(******ErrorStatus******)
IF axisdata[4].Axis_Error OR axisdata[5].Axis_Error THEN
	FeedIndexer.ErrorStatus.errErrorActive:=1;
ELSE
	FeedIndexer.ErrorStatus.errErrorActive:=0;
END_IF
FeedIndexer.ErrorStatus.errFieldBus:=0;
FeedIndexer.ErrorStatus.errLim2CCW:=b_limit_final_ccw_FI;
FeedIndexer.ErrorStatus.errLim2CW:=b_limit_final_cw_FI;
IF status_code4 = 'E2059' OR status_code5 = 'E2059' THEN
	FeedIndexer.ErrorStatus.errLimV_Err:=1;
ELSE
	FeedIndexer.ErrorStatus.errLimV_Err:=0;
END_IF
FeedIndexer.ErrorStatus.errMotComm:=(NOT(axisdata[4].Axis_NRT) OR NOT(axisdata[5].Axis_NRT));
IF status_code4 = 'F2031' OR status_code5 = 'F2031' THEN
	FeedIndexer.ErrorStatus.errMotEnc:=1;
ELSE
	FeedIndexer.ErrorStatus.errMotEnc:=0;
END_IF
IF status_code4 = 'F2021' OR status_code5 = 'F2021' OR FeedIndexer.ErrorStatus.errMotEnc THEN
	FeedIndexer.ErrorStatus.errMotor:=1;
ELSE
	FeedIndexer.ErrorStatus.errMotor:=0;
END_IF
IF FeedIndexer.ErrorStatus.errMotor OR FeedIndexer.ErrorStatus.errMotEnc THEN
	FeedIndexer.ErrorStatus.errMotReady:=1;
ELSE
	FeedIndexer.ErrorStatus.errMotReady:=0;
END_IF
FeedIndexer.ErrorStatus.errOverride:=0;
FeedIndexer.ErrorStatus.errV_DevExceed:=FeedIndexer.ErrorStatus.errLimV_Err;
IF status_code4 = 'F2075' THEN
	FeedIndexer.ErrorStatus.errP_RangeExceed:=1;
ELSE
	FeedIndexer.ErrorStatus.errP_RangeExceed:=0;
END_IF
IF status_code4 = 'F2037' OR status_code5 = 'F2037' THEN
	FeedIndexer.ErrorStatus.errP_DevExceed:=1;
ELSE
	FeedIndexer.ErrorStatus.errP_DevExceed:=0;
END_IF
FeedIndexer.ErrorStatus.errPosEnc:=FeedIndexer.Status.encBoxOp;
FeedIndexer.ErrorStatus.errPosEnc_Fo:=FeedIndexer.Status.encBoxOp;
IF status_code4 = 'F2026' OR status_code5 = 'F2026' THEN
	FeedIndexer.ErrorStatus.errPower:=1;
ELSE
	FeedIndexer.ErrorStatus.errPower:=0;
END_IF
(***** Error status end*****)


(*******Warning state********)
FeedIndexer.WarningStatus.waLim1CW:=b_limit_cw_FI;
FeedIndexer.WarningStatus.waLim1CCW:=b_limit_ccw_FI;
IF status_code4 = 'E8029' OR status_code5 = 'E8029' THEN
	FeedIndexer.WarningStatus.waLimSoftCW:=1;
ELSE
	FeedIndexer.WarningStatus.waLimSoftCW:=0;
END_IF
IF status_code4 = 'E8030' OR status_code5 = 'E8030' THEN
	FeedIndexer.WarningStatus.waLimSoftCCW:=1;
ELSE
	FeedIndexer.WarningStatus.waLimSoftCCW:=0;
END_IF
IF status_code4 = 'E8260' OR status_code5 = 'E8260' THEN
	FeedIndexer.WarningStatus.waMmaxExceeded:=1;
ELSE
	FeedIndexer.WarningStatus.waMmaxExceeded:=0;
END_IF
FeedIndexer.WarningStatus.waMotReady:=FeedIndexer.ErrorStatus.errMotReady;
FeedIndexer.WarningStatus.waMotWarn:=(axisdata[4].Axis_Warning OR axisdata[4].Axis_Warning);
FeedIndexer.WarningStatus.waOverride:=0;
FeedIndexer.WarningStatus.waParamFault:=(FeedIndexer.WarningStatus.waMotReady OR FeedIndexer.ErrorStatus.errMotReady);
IF status_code4 = 'E2031' OR status_code5 = 'E2031' THEN
	FeedIndexer.WarningStatus.waPosEncWarn:=1;
ELSE
	FeedIndexer.WarningStatus.waPosEncWarn:=0;
END_IF
FeedIndexer.WarningStatus.waStowPinsDep:=FALSE;
FeedIndexer.WarningStatus.waVelLimit:=FeedIndexer.ErrorStatus.errV_DevExceed;
(*********Warning status end***********)
(*****motor1****)
FeedIndexer.MotorOne.ErrorCode:= STRING_TO_UINT(status_code4);
FeedIndexer.MotorOne.mActTorq:=r_torque_4*7.1;
FeedIndexer.MotorOne.mActVelocity:=i_speed_4;
FeedIndexer.MotorOne.MotorTemp:=r_temp_motor4;
FeedIndexer.MotorOne.RateOfUtil:=r_torque_4;
FeedIndexer.MotorOne.MotorOverload:=r_torque_4;
(*****motor2****)
FeedIndexer.MotorTwo.ErrorCode:= STRING_TO_UINT(status_code5);
FeedIndexer.MotorTwo.mActTorq:=r_torque_5*7.1;
FeedIndexer.MotorTwo.mActVelocity:=i_speed_5;
FeedIndexer.MotorTwo.MotorTemp:=r_temp_motor5;
FeedIndexer.MotorTwo.RateOfUtil:=r_torque_5;
FeedIndexer.MotorTwo.MotorOverload:=r_torque_5;

END_PROGRAM

// IndraMotionMlc1/Application/POUs/OPCUA/OPCUA_Node/P_Opcua_Safety
PROGRAM P_Opcua_Safety
VAR
	b_final_limit_active:BOOL;
	fb_move_stow_Az: MC_MoveAbsolute;
	fb_move_stow_El: MC_MoveAbsolute;
	fb_ton_stow: TON;
	fb_self_reset_stow: R_Trig;
	fb_ton_self_reset_stow: TON;
	fb_rtrig_off_stow:R_Trig;
	fb_rtrig_lock_stow: R_Trig;
	fb_rtrig_reset_deploy: R_Trig;
	fb_rtrig_reset_retract: R_Trig;
	fb_rtrig_estop: R_TRIG;
	fb_rtrig_interlock_Az: R_TRIG;
	fb_rtrig_interlock_El: R_TRIG;
	fb_rtrig_interlock_Fi: R_TRIG;
	
	fb_ton_sim_stow: TON;
	_retract: TON;
	fb_ton_sim_retract: TON;
	fb_ton_sim_deploy: TON;
	fb_rtrig_sim_retract: R_TRIG;
	fb_rtrig_sim_deploy: R_TRIG;
	fb_rtrig_stow_deactivate: R_TRIG;
	fb_rtrig_stow_pulse: R_TRIG;
	_test: BOOL;
	b_stow_SIP: BOOL;
	rtrig_Estop_Az: R_TRIG;
	fb_Estop_Az: MC_Stop;
	rtrig_Estop_El: R_TRIG;
	fb_Estop_El: MC_Stop;
	rtrig_Estop_Fi: R_TRIG;
	fb_Estop_Fi: MC_Stop;
	MC_MoveRelative_0: MC_MoveRelative;
	MC_MoveRelative_1: MC_MoveRelative;
	R_TRIG_0: R_TRIG;
	TON_0: TON;
	b_stow_wait: BOOL;
	TON_1: TON;
	b_stow_run: BOOL;
	R_TRIG_1: R_TRIG;
	F_TRIG_0: F_TRIG;
	F_TRIG_1: F_TRIG;
	F_TRIG_2: F_TRIG;
	F_TRIG_3: F_TRIG;
	F_TRIG_4: F_TRIG;
	fb_rtrig_deactivate_El: R_TRIG;
	fb_rtrig_clear_stow: R_TRIG;
	F_TRIG_5: F_trig;
END_VAR
VAR // added by the converter: edge detectors and wires of the graphical bodies
    _w1, _w2, _w3, _w4, _w5, _w6 : BOOL;
END_VAR

safety();
(*IF b_HHP_Estop OR b_Turnhead_Estop OR b_DS_Estop OR b_FI_Estop OR b_Turnhead_Hatch OR b_AZ_Hatch OR (NOT(b_stow_pin_limit_unlock)) THEN
	b_in_interlock:=1;
ELSE
	b_in_interlock:=0;
END_IF*)

(*IF b_in_interlock OR b_DSDoor_Estop OR b_PSCDoor_Estop OR b_DriveCabinetDoor_Estop OR b_EMISCDoor_Estop THEN // b_in_interlock true will cause an EStop. Whereas it should only cause an interlock. 
	b_in_Estop:=1;
ELSE
	b_in_Estop:=0;
END_IF*)
safety.Status.AutoStowActive:=0;
safety.Status.Axes_InitFault:=NOT(Azimuth.Status.InitOk AND Elevation.Status.InitOk AND FeedIndexer.Status.InitOk);
safety.Status.EStopFi:=b_FI_Estop;
safety.Status.EStopHHP:=b_HHP_Estop;
safety.Status.EStopPED:=b_DS_Estop;
safety.Status.EStopTurnhead:=b_Turnhead_Estop;
safety.Status.HatchTurnheadRoof:=b_Turnhead_Hatch;
safety.Status.HatchAzBearing:=b_AZ_Hatch;
//safety.InterlockAck
safety.Status.Lim2_CCW_Az:=b_limit_final_ccw_az;
safety.Status.Lim2_CCW_Fi:=b_limit_final_ccw_Fi;
safety.Status.Lim2_CW_Az:=b_limit_final_cw_az;
safety.Status.Lim2_CW_Fi:=b_limit_final_cw_Fi;
safety.Status.Lim2_Dn_El:=b_limit_final_ccw_el;
safety.Status.Lim2_Up_El:=b_limit_final_cw_el;
b_final_limit_active:=(safety.Status.Lim2_CCW_Az OR safety.Status.Lim2_CW_Az OR safety.Status.Lim2_Dn_El OR safety.Status.Lim2_Up_El OR safety.Status.Lim2_CCW_Fi OR safety.Status.Lim2_CW_Fi); 

(* Still to be wired in *)
safety.Status.SafetyLockout_Az:=NOT(b_Lock_Out_Az);
safety.Status.SafetyLockout_El:=NOT(b_Lock_Out_El);
safety.Status.SafetyLockout_Fi:=NOT(b_Lock_Out_Fi);

IF safety.Status.Axes_InitFault THEN
	safety.Status.SafetyState:=SafetyStatetype.Stopped;
ELSIF b_in_interlock OR b_in_Estop OR b_final_limit_active THEN
	safety.Status.SafetyState:=SafetyStatetype.Error;
ELSE
	safety.Status.SafetyState:=SafetyStatetype.Running;	
END_IF
safety.Status.STO_Az:=b_in_interlock;
safety.Status.STO_El:=b_in_interlock;
safety.Status.STO_Fi:=b_in_interlock;

IF b_stow_pin_deploy AND NOT(b_stow_pin_limit_lock) THEN
	safety.Status.StowPinStatus:=StowPinStatustype.Deploying;
ELSIF b_stow_pin_limit_lock THEN
	safety.Status.StowPinStatus:=StowPinStatustype.Deployed;
ELSIF b_stow_pin_retract AND NOT(b_stow_pin_limit_unlock) THEN
	safety.Status.StowPinStatus:=StowPinStatustype.Retracting;
ELSIF NOT(b_stow_pin_limit_unlock) THEN
	safety.Status.StowPinStatus:=StowPinStatustype.Retracted;
END_IF

IF (Azimuth.Status.p_Enc >= Azimuth.Status.StowPos_Minus AND Azimuth.Status.p_Enc <= Azimuth.Status.StowPos_Plus) THEN
	b_stow_lock_allow:=1;
ELSE 
	b_stow_lock_allow:=0;
END_IF

(*
IF b_in_interlock AND b_in_Estop THEN 
	Safety.Status.InterlockClearable:=0;
ELSE
	Safety.Status.InterlockClearable:=1;	
END_IF *)

// Run Ladder Logic
P_Opcua_Safety.A_STOW();
P_Opcua_Safety.A_Interlock_Estop();

ACTION A_STOW:
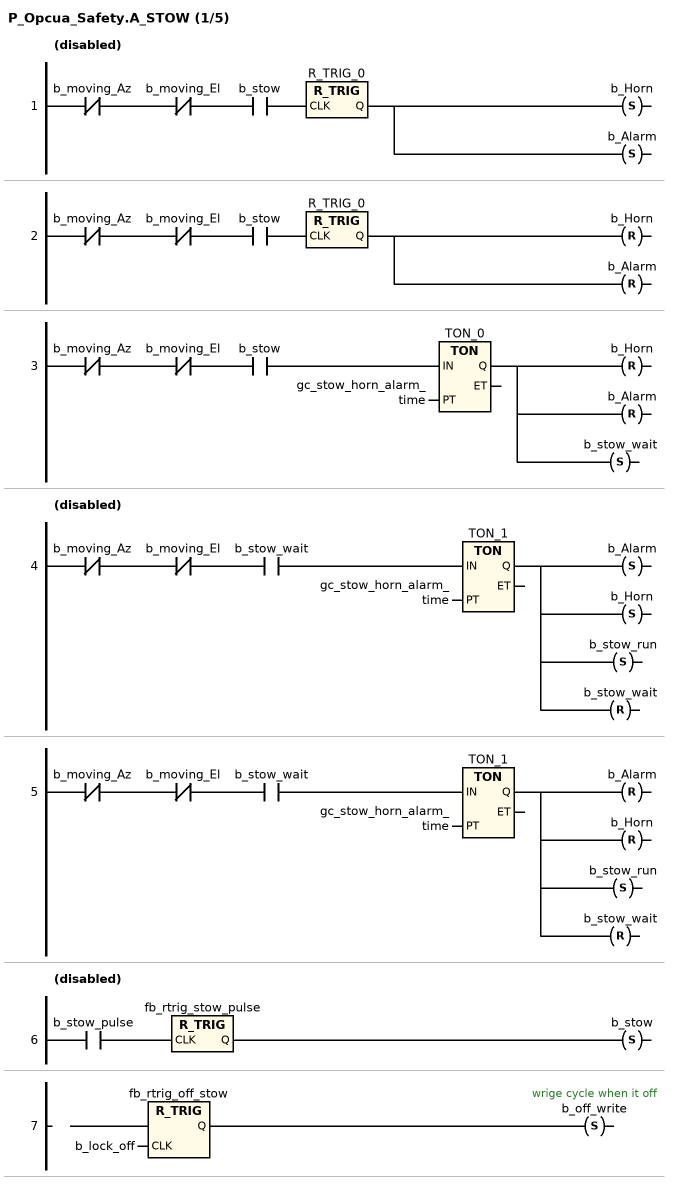
// NETWORK 1 (disabled)
// R_TRIG_0(CLK := NOT b_moving_Az AND NOT b_moving_El AND b_stow); // R_TRIG
// b_Horn S= R_TRIG_0.Q;
// b_Alarm S= R_TRIG_0.Q;

// NETWORK 2
R_TRIG_0(CLK := NOT b_moving_Az AND NOT b_moving_El AND b_stow); // R_TRIG
b_Horn R= R_TRIG_0.Q;
b_Alarm R= R_TRIG_0.Q;

// NETWORK 3
TON_0(IN := NOT b_moving_Az AND NOT b_moving_El AND b_stow, PT := gc_stow_horn_alarm_time); // TON
b_Horn R= TON_0.Q;
b_Alarm R= TON_0.Q;
b_stow_wait S= TON_0.Q;

// NETWORK 4 (disabled)
// TON_1(IN := NOT b_moving_Az AND NOT b_moving_El AND b_stow_wait, PT := gc_stow_horn_alarm_time); // TON
// b_Alarm S= TON_1.Q;
// b_Horn S= TON_1.Q;
// b_stow_run S= TON_1.Q;
// b_stow_wait R= TON_1.Q;

// NETWORK 5
TON_1(IN := NOT b_moving_Az AND NOT b_moving_El AND b_stow_wait, PT := gc_stow_horn_alarm_time); // TON
b_Alarm R= TON_1.Q;
b_Horn R= TON_1.Q;
b_stow_run S= TON_1.Q;
b_stow_wait R= TON_1.Q;

// NETWORK 6 (disabled)
//   fb_rtrig_stow_pulse: the definition of rise trigger,The function block R_TRIG detects a rising edge.
// fb_rtrig_stow_pulse(CLK := b_stow_pulse); // R_TRIG
// b_stow S= fb_rtrig_stow_pulse.Q;

// NETWORK 7
//   b_lock_off: power off after arriving at the stow position
//   b_off_write: wrige cycle when it off
fb_rtrig_off_stow(CLK := b_lock_off); // R_TRIG
b_off_write S= fb_rtrig_off_stow.Q;

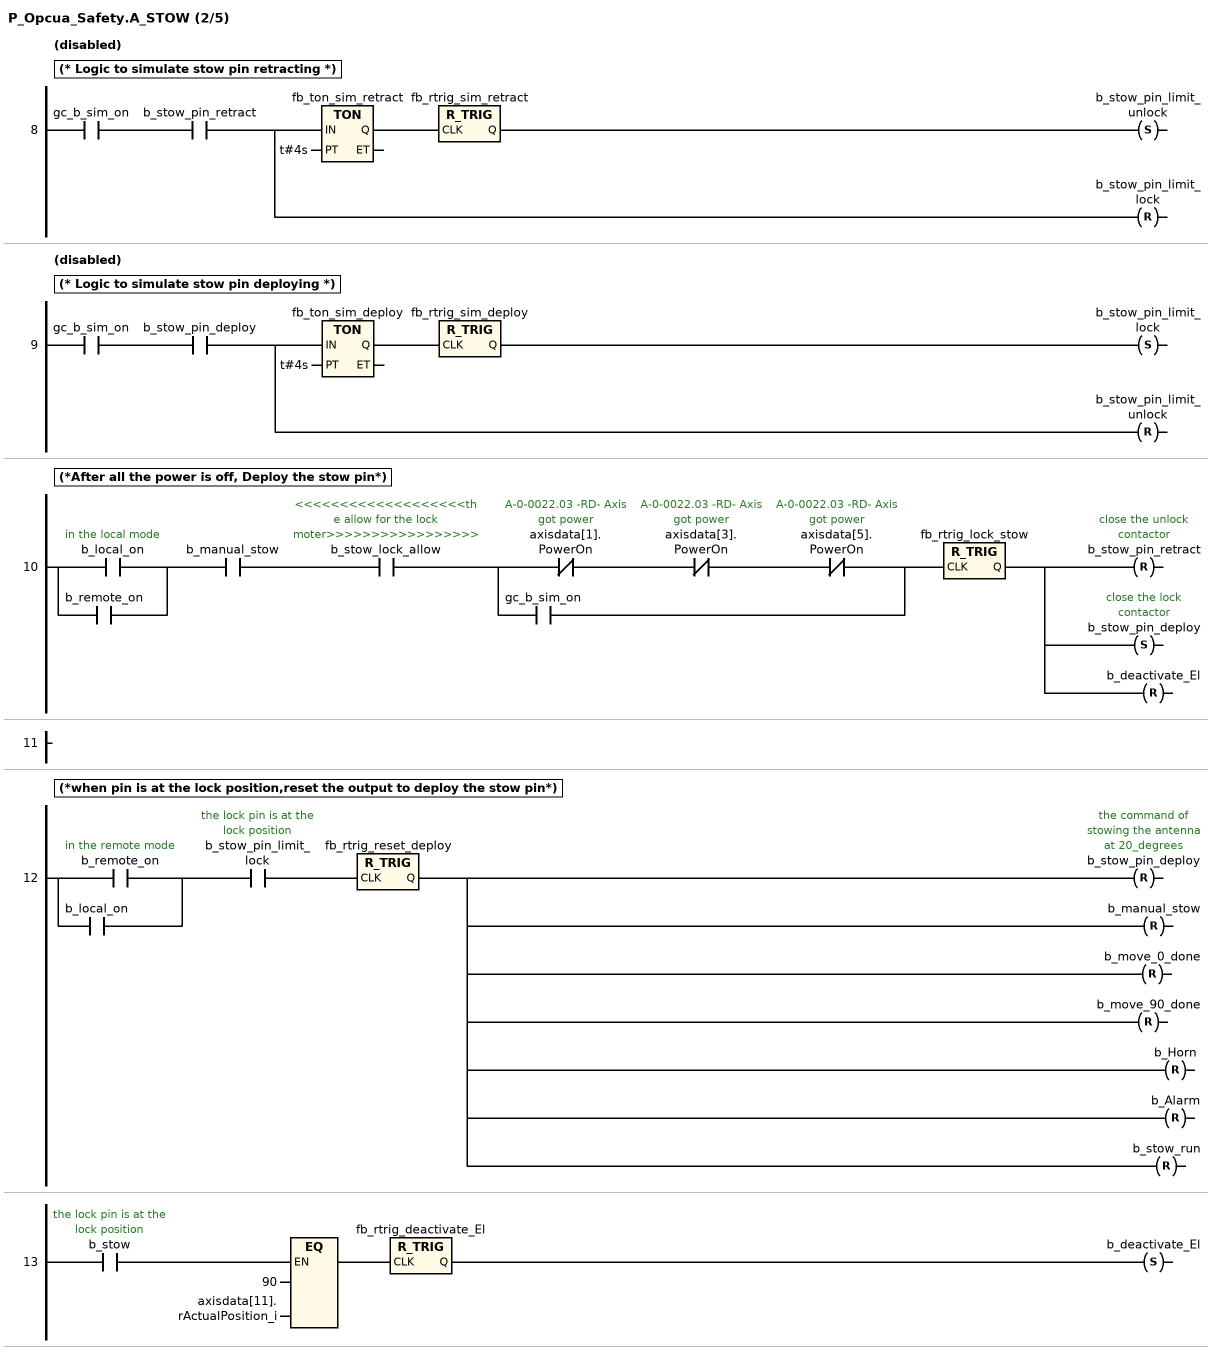
// NETWORK 8 (disabled)
//   fb_rtrig_sim_retract: the definition of rise trigger,The function block R_TRIG detects a rising edge.
//   fb_ton_sim_retract: The function block Timer On Delay implements a turn-on delay
// label: (* Logic to simulate stow pin retracting *)
// _w1 := gc_b_sim_on AND b_stow_pin_retract;
// fb_ton_sim_retract(IN := _w1, PT := t#4s); // TON
// fb_rtrig_sim_retract(CLK := fb_ton_sim_retract.Q); // R_TRIG
// b_stow_pin_limit_unlock S= fb_rtrig_sim_retract.Q;
// b_stow_pin_limit_lock R= _w1;

// NETWORK 9 (disabled)
//   fb_rtrig_sim_deploy: the definition of rise trigger,The function block R_TRIG detects a rising edge.
//   fb_ton_sim_deploy: The function block Timer On Delay implements a turn-on delay
// label: (* Logic to simulate stow pin deploying *)
// _w2 := gc_b_sim_on AND b_stow_pin_deploy;
// fb_ton_sim_deploy(IN := _w2, PT := t#4s); // TON
// fb_rtrig_sim_deploy(CLK := fb_ton_sim_deploy.Q); // R_TRIG
// b_stow_pin_limit_lock S= fb_rtrig_sim_deploy.Q;
// b_stow_pin_limit_unlock R= _w2;

// NETWORK 10
//   fb_rtrig_lock_stow: the definition of rise trigger,The function block R_TRIG detects a rising edge.
//   b_local_on: in the local mode
//   b_stow_lock_allow: <<<<<<<<<<<<<<<<<<<the allow for the lock moter>>>>>>>>>>>>>>>>>
//   axisdata[1].PowerOn: A-0-0022.03 -RD- Axis got power
//   axisdata[3].PowerOn: A-0-0022.03 -RD- Axis got power
//   axisdata[5].PowerOn: A-0-0022.03 -RD- Axis got power
//   b_stow_pin_retract: close the unlock contactor
//   b_stow_pin_deploy: close the lock contactor
// label: (*After all the power is off, Deploy the stow pin*)
fb_rtrig_lock_stow(CLK := (b_local_on OR b_remote_on) AND b_manual_stow AND b_stow_lock_allow AND (NOT axisdata[1].PowerOn AND NOT axisdata[3].PowerOn AND NOT axisdata[5].PowerOn OR gc_b_sim_on)); // R_TRIG
b_stow_pin_retract R= fb_rtrig_lock_stow.Q;
b_stow_pin_deploy S= fb_rtrig_lock_stow.Q;
b_deactivate_El R= fb_rtrig_lock_stow.Q;

// NETWORK 11

// NETWORK 12
//   b_remote_on: in the remote mode
//   b_stow_pin_limit_lock: the lock pin is at the lock position
//   b_stow_pin_deploy: the command of stowing the antenna at 20_degrees
// label: (*when pin is at the lock position,reset the output to deploy the stow pin*)
fb_rtrig_reset_deploy(CLK := (b_remote_on OR b_local_on) AND b_stow_pin_limit_lock); // R_TRIG
b_stow_pin_deploy R= fb_rtrig_reset_deploy.Q;
b_manual_stow R= fb_rtrig_reset_deploy.Q;
b_move_0_done R= fb_rtrig_reset_deploy.Q;
b_move_90_done R= fb_rtrig_reset_deploy.Q;
b_Horn R= fb_rtrig_reset_deploy.Q;
b_Alarm R= fb_rtrig_reset_deploy.Q;
b_stow_run R= fb_rtrig_reset_deploy.Q;

// NETWORK 13
//   b_stow: the lock pin is at the lock position
fb_rtrig_deactivate_El(CLK := b_stow AND 90 = axisdata[11].rActualPosition_i); // R_TRIG
b_deactivate_El S= fb_rtrig_deactivate_El.Q;

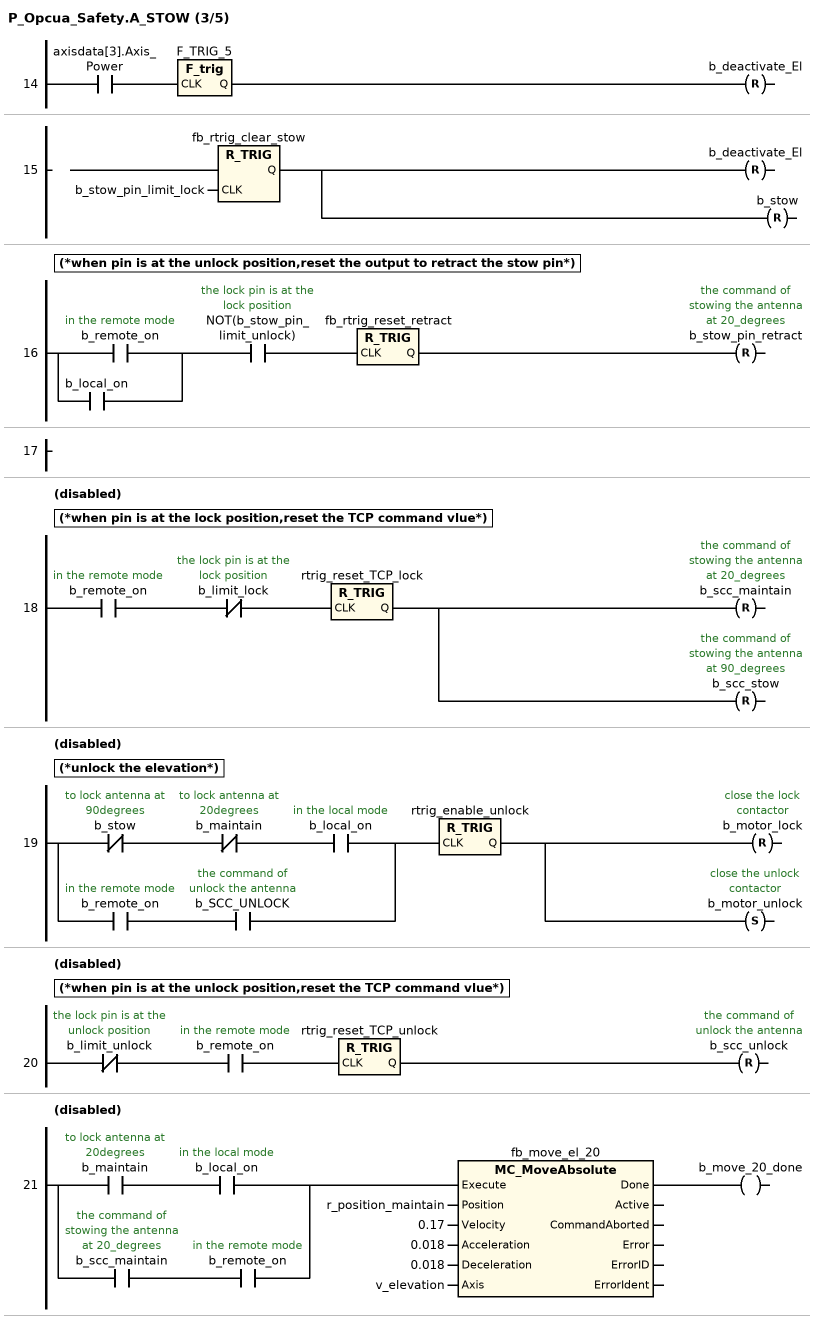
// NETWORK 14
F_TRIG_5(CLK := axisdata[3].Axis_Power); // F_trig
b_deactivate_El R= F_TRIG_5.Q;

// NETWORK 15
//   b_stow_pin_limit_lock: the lock pin is at the lock position
fb_rtrig_clear_stow(CLK := b_stow_pin_limit_lock); // R_TRIG
b_deactivate_El R= fb_rtrig_clear_stow.Q;
b_stow R= fb_rtrig_clear_stow.Q;

// NETWORK 16
//   b_remote_on: in the remote mode
//   NOT(b_stow_pin_limit_unlock): the lock pin is at the lock position
//   b_stow_pin_retract: the command of stowing the antenna at 20_degrees
// label: (*when pin is at the unlock position,reset the output to retract the stow pin*)
fb_rtrig_reset_retract(CLK := (b_remote_on OR b_local_on) AND (NOT(b_stow_pin_limit_unlock))); // R_TRIG
b_stow_pin_retract R= fb_rtrig_reset_retract.Q;

// NETWORK 17

// NETWORK 18 (disabled)
//   b_remote_on: in the remote mode
//   b_limit_lock: the lock pin is at the lock position
//   b_scc_maintain: the command of stowing the antenna at 20_degrees
//   b_scc_stow: the command of stowing the antenna at 90_degrees
// label: (*when pin is at the lock position,reset the TCP command vlue*)
// rtrig_reset_TCP_lock(CLK := b_remote_on AND NOT b_limit_lock); // R_TRIG
// b_scc_maintain R= rtrig_reset_TCP_lock.Q;
// b_scc_stow R= rtrig_reset_TCP_lock.Q;

// NETWORK 19 (disabled)
//   b_stow: to lock antenna at 90degrees
//   b_maintain: to lock antenna at 20degrees
//   b_local_on: in the local mode
//   b_remote_on: in the remote mode
//   b_SCC_UNLOCK: the command of unlock the antenna
//   b_motor_lock: close the lock contactor
//   b_motor_unlock: close the unlock contactor
// label: (*unlock the elevation*)
// rtrig_enable_unlock(CLK := NOT b_stow AND NOT b_maintain AND b_local_on OR b_remote_on AND b_SCC_UNLOCK); // R_TRIG
// b_motor_lock R= rtrig_enable_unlock.Q;
// b_motor_unlock S= rtrig_enable_unlock.Q;

// NETWORK 20 (disabled)
//   b_limit_unlock: the lock pin is at the unlock position
//   b_remote_on: in the remote mode
//   b_scc_unlock: the command of unlock the antenna
// label: (*when pin is at the unlock position,reset the TCP command vlue*)
// rtrig_reset_TCP_unlock(CLK := NOT b_limit_unlock AND b_remote_on); // R_TRIG
// b_scc_unlock R= rtrig_reset_TCP_unlock.Q;

// NETWORK 21 (disabled)
//   b_maintain: to lock antenna at 20degrees
//   b_local_on: in the local mode
//   b_scc_maintain: the command of stowing the antenna at 20_degrees
//   b_remote_on: in the remote mode
//   v_elevation: Virtual axis "v_elevation" with axis number 8
// fb_move_el_20(
//     Execute := b_maintain AND b_local_on OR b_scc_maintain AND b_remote_on,
//     Position := r_position_maintain,
//     Velocity := 0.17,
//     Acceleration := 0.018,
//     Deceleration := 0.018,
//     Axis := v_elevation); // MC_MoveAbsolute
// b_move_20_done := fb_move_el_20.Done;

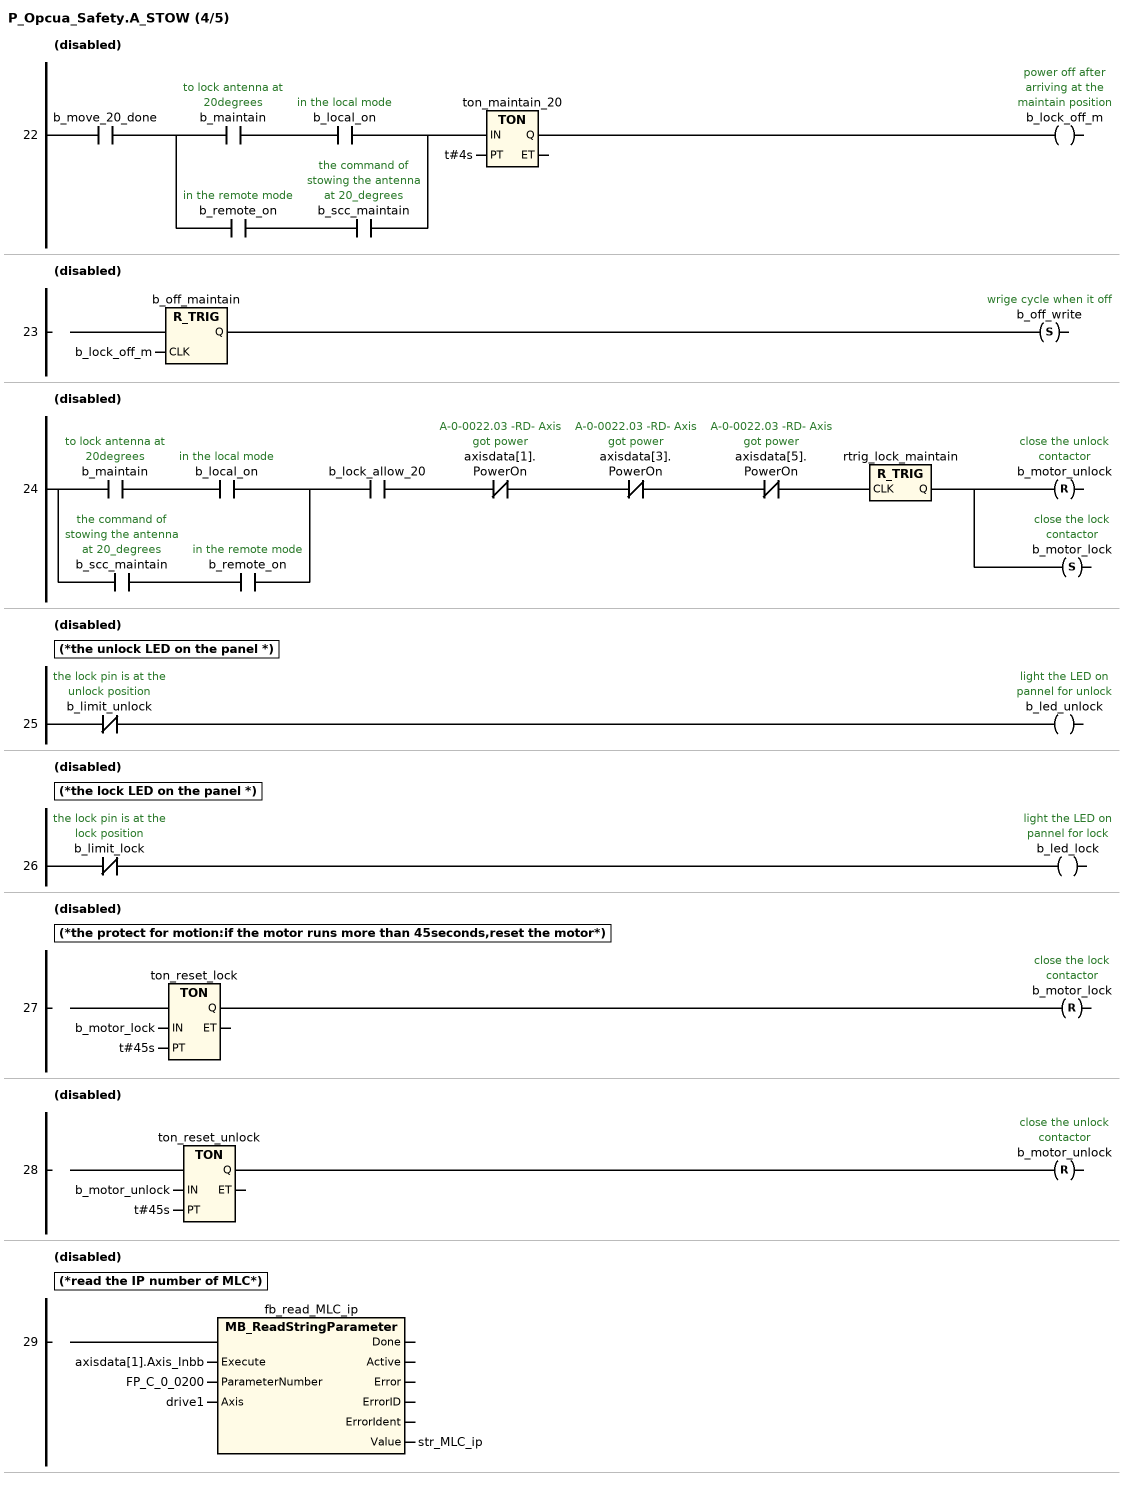
// NETWORK 22 (disabled)
//   b_maintain: to lock antenna at 20degrees
//   b_local_on: in the local mode
//   b_remote_on: in the remote mode
//   b_scc_maintain: the command of stowing the antenna at 20_degrees
//   b_lock_off_m: power off after arriving at the maintain position
// ton_maintain_20(IN := b_move_20_done AND (b_maintain AND b_local_on OR b_remote_on AND b_scc_maintain), PT := t#4s); // TON
// b_lock_off_m := ton_maintain_20.Q;

// NETWORK 23 (disabled)
//   b_lock_off_m: power off after arriving at the maintain position
//   b_off_write: wrige cycle when it off
// b_off_maintain(CLK := b_lock_off_m); // R_TRIG
// b_off_write S= b_off_maintain.Q;

// NETWORK 24 (disabled)
//   b_maintain: to lock antenna at 20degrees
//   b_local_on: in the local mode
//   b_scc_maintain: the command of stowing the antenna at 20_degrees
//   b_remote_on: in the remote mode
//   axisdata[1].PowerOn: A-0-0022.03 -RD- Axis got power
//   axisdata[3].PowerOn: A-0-0022.03 -RD- Axis got power
//   axisdata[5].PowerOn: A-0-0022.03 -RD- Axis got power
//   b_motor_unlock: close the unlock contactor
//   b_motor_lock: close the lock contactor
// rtrig_lock_maintain(CLK := (b_maintain AND b_local_on OR b_scc_maintain AND b_remote_on) AND b_lock_allow_20 AND NOT axisdata[1].PowerOn AND NOT axisdata[3].PowerOn AND NOT axisdata[5].PowerOn); // R_TRIG
// b_motor_unlock R= rtrig_lock_maintain.Q;
// b_motor_lock S= rtrig_lock_maintain.Q;

// NETWORK 25 (disabled)
//   b_limit_unlock: the lock pin is at the unlock position
//   b_led_unlock: light the LED on pannel for unlock
// label: (*the unlock LED on the panel *)
// b_led_unlock := NOT b_limit_unlock;

// NETWORK 26 (disabled)
//   b_limit_lock: the lock pin is at the lock position
//   b_led_lock: light the LED on pannel for lock
// label: (*the lock LED on the panel *)
// b_led_lock := NOT b_limit_lock;

// NETWORK 27 (disabled)
//   b_motor_lock: close the lock contactor
// label: (*the protect for motion:if the motor runs more than 45seconds,reset the motor*)
// ton_reset_lock(IN := b_motor_lock, PT := t#45s); // TON
// b_motor_lock R= ton_reset_lock.Q;

// NETWORK 28 (disabled)
//   b_motor_unlock: close the unlock contactor
// ton_reset_unlock(IN := b_motor_unlock, PT := t#45s); // TON
// b_motor_unlock R= ton_reset_unlock.Q;

// NETWORK 29 (disabled)
//   axisdata[1].Axis_Inbb: A-0-0021.13 -RD- Axis is ready for power to the amplifier (bb)
//   FP_C_0_0200: Engineering, IP address
//   drive1: Real axis "Drive1" with axis number 1
//   str_MLC_ip: IP number in MLC
// label: (*read the IP number of MLC*)
// fb_read_MLC_ip(
//     Execute := axisdata[1].Axis_Inbb,
//     ParameterNumber := FP_C_0_0200,
//     Axis := drive1,
//     Value => str_MLC_ip); // MB_ReadStringParameter

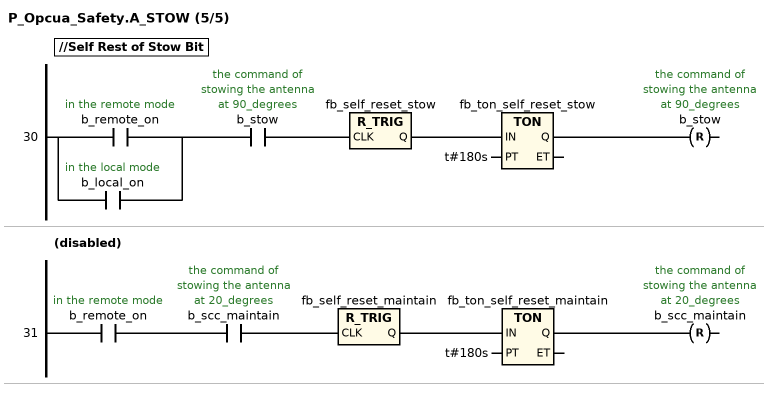
// NETWORK 30
//   b_remote_on: in the remote mode
//   b_local_on: in the local mode
//   b_stow: the command of stowing the antenna at 90_degrees
// label: //Self Rest of Stow Bit
fb_self_reset_stow(CLK := (b_remote_on OR b_local_on) AND b_stow); // R_TRIG
fb_ton_self_reset_stow(IN := fb_self_reset_stow.Q, PT := t#180s); // TON
b_stow R= fb_ton_self_reset_stow.Q;

// NETWORK 31 (disabled)
//   b_remote_on: in the remote mode
//   b_scc_maintain: the command of stowing the antenna at 20_degrees
// fb_self_reset_maintain(CLK := b_remote_on AND b_scc_maintain); // R_TRIG
// fb_ton_self_reset_maintain(IN := fb_self_reset_maintain.Q, PT := t#180s); // TON
// b_scc_maintain R= fb_ton_self_reset_maintain.Q;
END_ACTION

ACTION A_Interlock_Estop:
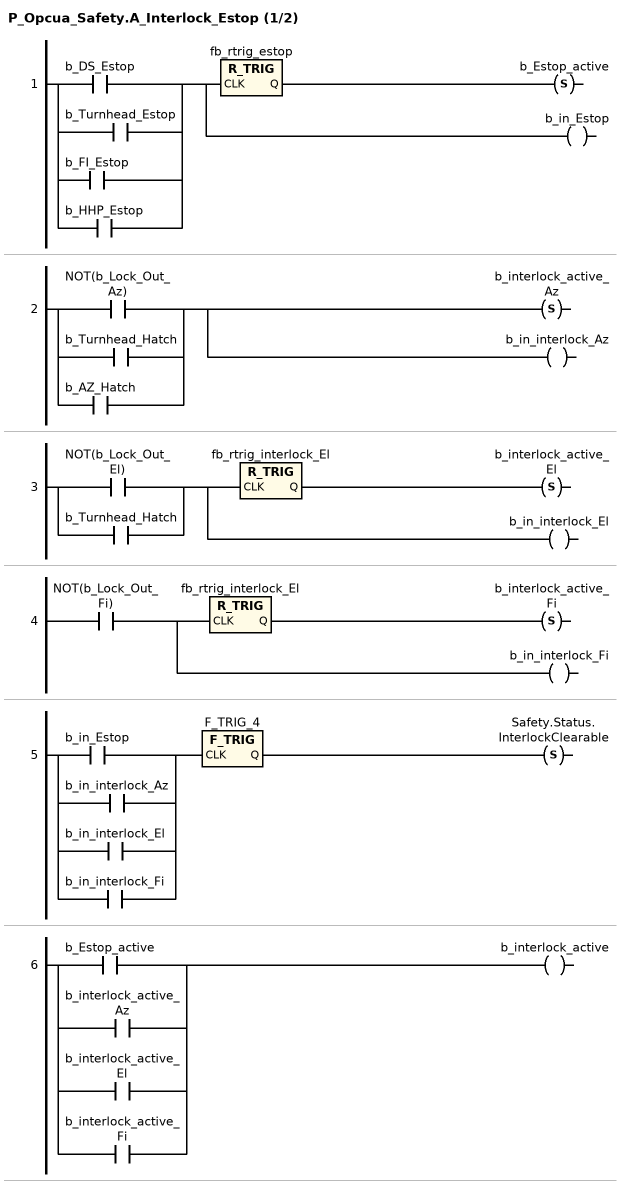
// NETWORK 1
_w3 := b_DS_Estop OR b_Turnhead_Estop OR b_FI_Estop OR b_HHP_Estop;
fb_rtrig_estop(CLK := _w3); // R_TRIG
b_Estop_active S= fb_rtrig_estop.Q;
b_in_Estop := _w3;

// NETWORK 2
_w4 := (NOT(b_Lock_Out_Az)) OR b_Turnhead_Hatch OR b_AZ_Hatch;
b_interlock_active_Az S= _w4;
b_in_interlock_Az := _w4;

// NETWORK 3
_w5 := (NOT(b_Lock_Out_El)) OR b_Turnhead_Hatch;
fb_rtrig_interlock_El(CLK := _w5); // R_TRIG
b_interlock_active_El S= fb_rtrig_interlock_El.Q;
b_in_interlock_El := _w5;

// NETWORK 4
_w6 := NOT(b_Lock_Out_Fi);
fb_rtrig_interlock_El(CLK := _w6); // R_TRIG
b_interlock_active_Fi S= fb_rtrig_interlock_El.Q;
b_in_interlock_Fi := _w6;

// NETWORK 5
F_TRIG_4(CLK := b_in_Estop OR b_in_interlock_Az OR b_in_interlock_El OR b_in_interlock_Fi); // F_TRIG
Safety.Status.InterlockClearable S= F_TRIG_4.Q;

// NETWORK 6
b_interlock_active := b_Estop_active OR b_interlock_active_Az OR b_interlock_active_El OR b_interlock_active_Fi;

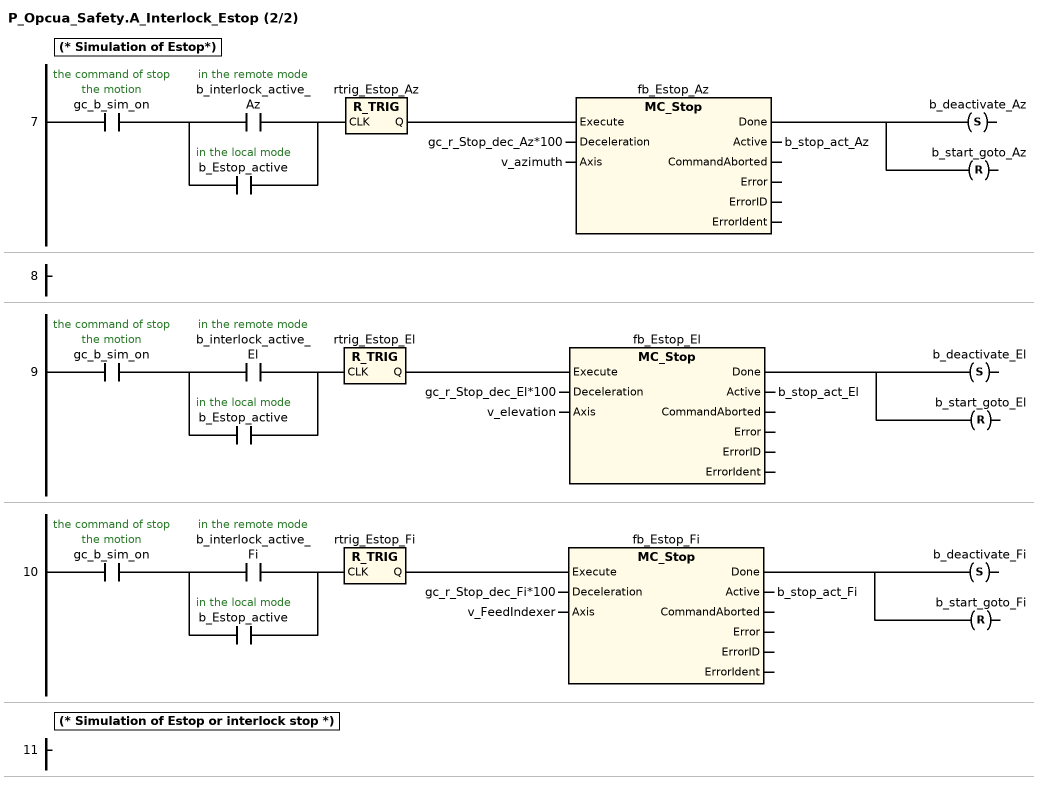
// NETWORK 7
//   gc_b_sim_on: the command of stop the motion
//   b_interlock_active_Az: in the remote mode
//   b_Estop_active: in the local mode
//   v_azimuth: Virtual axis "v_azimuth" with axis number 7
// label: (* Simulation of Estop*)
rtrig_Estop_Az(CLK := gc_b_sim_on AND (b_interlock_active_Az OR b_Estop_active)); // R_TRIG
fb_Estop_Az(
    Execute := rtrig_Estop_Az.Q,
    Deceleration := gc_r_Stop_dec_Az*100,
    Axis := v_azimuth,
    Active => b_stop_act_Az); // MC_Stop
b_deactivate_Az S= fb_Estop_Az.Done;
b_start_goto_Az R= fb_Estop_Az.Done;

// NETWORK 8

// NETWORK 9
//   gc_b_sim_on: the command of stop the motion
//   b_interlock_active_El: in the remote mode
//   b_Estop_active: in the local mode
//   v_elevation: Virtual axis "v_elevation" with axis number 8
rtrig_Estop_El(CLK := gc_b_sim_on AND (b_interlock_active_El OR b_Estop_active)); // R_TRIG
fb_Estop_El(
    Execute := rtrig_Estop_El.Q,
    Deceleration := gc_r_Stop_dec_El*100,
    Axis := v_elevation,
    Active => b_stop_act_El); // MC_Stop
b_deactivate_El S= fb_Estop_El.Done;
b_start_goto_El R= fb_Estop_El.Done;

// NETWORK 10
//   gc_b_sim_on: the command of stop the motion
//   b_interlock_active_Fi: in the remote mode
//   b_Estop_active: in the local mode
//   v_FeedIndexer: Virtual axis "v_polarization" with axis number 9
rtrig_Estop_Fi(CLK := gc_b_sim_on AND (b_interlock_active_Fi OR b_Estop_active)); // R_TRIG
fb_Estop_Fi(
    Execute := rtrig_Estop_Fi.Q,
    Deceleration := gc_r_Stop_dec_Fi*100,
    Axis := v_FeedIndexer,
    Active => b_stop_act_Fi); // MC_Stop
b_deactivate_Fi S= fb_Estop_Fi.Done;
b_start_goto_Fi R= fb_Estop_Fi.Done;

// NETWORK 11
// label: (* Simulation of Estop or interlock stop *)
END_ACTION

END_PROGRAM

// IndraMotionMlc1/Application/POUs/OPCUA/OPCUA_Node/P_Opcua_CommandArbiter
PROGRAM P_Opcua_CommandArbiter
VAR
	cmds: CmdResponseType;
END_VAR

CommandArbiter();
//CommandArbiter.Status.DscCmdAuthority;


(* if hhp connected then 
    CommandArbiter.DscCmdAuthority:= HHP;
	End *)

END_PROGRAM

// IndraMotionMlc1/Application/POUs/OPCUA/OPCUA_Node/P_Opcua_Time_cds
PROGRAM P_Opcua_Time_cds
VAR
	IL_SysTime64_0: IL_SysTime64;
	Current_time: SYS_TIME64;
	UnixSeconds: Lreal;
	i_num_quarter_test: DINT;
	current_time_pos_test: LREAL;
	lr_MJD_Test: LREAL;
	
	dummy: Lreal;
	dummy2: BOOL;
	
END_VAR

Time_cds();
Current_time;
P_Opcua_Time_cds.Get_Time();
//Time_cds.Status.TAIOffset:=Current_time.HighValue*65536+Current_time.LowValue;
//Calculate TAI offset 
//Time_cds.Status.TAIOffset:=Current_time.HighValue*65536+Current_time.LowValue;
//Time_cds.Status.TAIOffset:=((Current_time.HighValue+4294967295)/1000000+ Current_time.LowValue/1000000);
UnixSeconds:=(TO_LREAL(Current_time.HighValue)*4294967295+TO_LREAL(Current_time.LowValue))/1000000; //UTC 
//Time_cds.Status.TAIOffset:=UnixSeconds-UnixToSKAEpoch-(Time_cds.Status.LeapSecPTP-Time_cds.Status.UTCtoSkaoEpochSec);

lr_MJD_Test:= UnixSeconds/86400+40587;

 // This should be the TAI offset after the SKAO epoch. The time from the Time Virtual axis.
//Time_cds.Status.DscTimeSyncSource:=Source_Timesync;

Time_cds.Status.LeapSecPTP:=LeapSecPTP;   
IF Source_Timesync = DscTimeSyncSourceType.PTP THEN
	Time_cds.Status.TimeSourceAddrNTP:=IP_Adress_PTP;
ELSIF Source_Timesync = DscTimeSyncSourceType.NTP THEN
	Time_cds.Status.TimeSourceAddrNTP:=IP_Adress_NTP;
ELSE
	Time_cds.Status.TimeSourceAddrNTP:=str_MLC_ip;
END_IF

IF Source_Timesync = DscTimeSyncSourceType.PTP THEN
	Time_cds.Status.TimeSynced:=b_M_time_done;
	b_no_SetDateTime:=FALSE;
ELSIF Source_Timesync = DscTimeSyncSourceType.NTP THEN
	//Time_cds.Status.TimeSynced:=b_M_time_done;
	b_no_SetDateTime:=FALSE;
ELSE	
    Time_cds.Status.TimeSynced:=b_M_time_done;
	// need to use system time to calculate MJD
	b_no_SetDateTime:=TRUE;
	
	di_MJD_day := LREAL_TO_DINT(TRUNC(UnixSeconds/86400+40587));
	i_num_quarter:=TRUNC((UnixSeconds-DINT_TO_LREAL(TRUNC(UnixSeconds/86400)*86400))/360);

 
	current_time_pos_test:=UnixSeconds-DINT_TO_LREAL(TRUNC(UnixSeconds/86400)*86400)-i_num_quarter*360;
	dummy:=axisdata[10].rActualPosition_i-current_time_pos_test;
	dummy2:=(ABS(dummy)>=0.10);
	IF (ABS(dummy)>=1.1 AND NOT(b_track_on)) THEN
//	current_time_pos:=current_time_pos_test;
//  	b_NTP_set_up:=TRUE;
	ELSE 
//	b_NTP_set_up:=FALSE;		
	END_IF
	
	
END_IF

ACTION Get_Time:
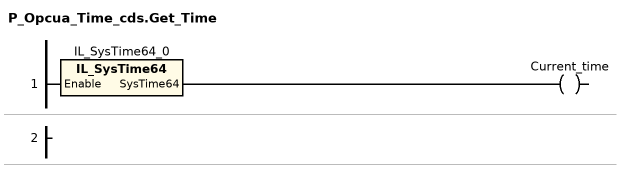
// NETWORK 1
IL_SysTime64_0(Enable := TRUE); // IL_SysTime64
Current_time := IL_SysTime64_0.SysTime64;

// NETWORK 2
END_ACTION

END_PROGRAM

// IndraMotionMlc1/Application/POUs/OPCUA/OPCUA_Node/P_Opcua_Management
PROGRAM P_Opcua_Management
VAR
	R_total_distance_AZ_old:LREAL;
	R_total_distance_EL_deg_old:LREAL;
	R_total_distance_EL_m_old:LREAL;
	R_total_distance_FI_old:LREAL;
	count_i:UINT;
	(*<<<<<<<<<<<<<<<<<<<<<<<<<<<<<<<<<<<< Stop >>>>>>>>>>>>>>>>>>>>>>>>>>>>>*)
	b_stop_Az_done: BOOL;
	b_stop_El_done: BOOL;
	b_stop_Fi_done: BOOL;
	fb_stop_Az: MC_Stop;
	fb_stop_El: MC_Stop;
	fb_stop_Fi: MC_Stop;
	rtrig_stop_Az: R_TRIG;
	rtrig_stop_El: R_TRIG;
	rtrig_stop_Fi: R_TRIG;
	rtrig_stop_stow: R_TRIG;
	rtrig_reset_stop: R_TRIG;
	
	(*<<<<<<<<<<<<<<<<<<<<<<<<<<<<<<<<<<<< Goto >>>>>>>>>>>>>>>>>>>>>>>>>>>>>*)
	// Az
	
	b_goto_done_Az: BOOL;
	b_active_Az:     BOOL;
	b_moving_Az: BOOL;
	fb_goto_Az: MC_MoveRelative;
	fb_start_goto_Az: R_Trig;
	fb_goto_done_Az : R_Trig;
	
	// El
	
	b_goto_done_El: BOOL;
	b_active_El:     BOOL;
	b_moving_El: BOOL;
	fb_goto_El: MC_MoveRelative;
	fb_start_goto_El: R_Trig;
	fb_goto_done_El : R_Trig;
	//Fi
	b_goto_done_Fi: BOOL;
	b_active_Fi:     BOOL;
	b_moving_Fi: BOOL;
	fb_goto_Fi: MC_MoveRelative;
	fb_start_goto_Fi: R_Trig;
	fb_goto_done_Fi : R_Trig;
	
(*<<<<<<<<<<<<<<<<<<<<<<<<<<<<<<<<<<<<<<<<<<<<<<<<<<<power>>>>>>>>>>>>>>>>>>>>>>>>>>>>>>>>>>>>*)
	ton_pow_off_Az: TON;
	ton_pow_off_El: TON;
	ton_pow_off_Fi: TON;
	rtrig_power_Az: R_TRIG;
	rtrig_power_El: R_TRIG;
	rtrig_power_Fi: R_TRIG;
	fb_ton_El: TON;
	fb_ton_Fi: TON;
	rtrig_off_Az: R_TRIG;
	rtrig_off_El: R_TRIG;
	rtrig_off_Fi: R_TRIG;
	rtrig_power_power: R_TRIG;
	b_pwr_on:BOOL;
	b_pwr_off: BOOL;
	b_clear_off_done_Az1: BOOL;
	b_clear_off_done_Az2: BOOL;
	b_clear_off_done_El: BOOL;
	b_clear_off_done_Fi1: BOOL;
	b_clear_off_done_Fi2: BOOL;
	
	FB_clear_error_off_Az1:MB_WriteParameter;
	FB_clear_error_off_Az2:MB_WriteParameter;
	FB_clear_error_off_El:MB_WriteParameter;
	FB_clear_error_off_Fi1:MB_WriteParameter;
	FB_clear_error_off_Fi2:MB_WriteParameter;
	rtrig_err: R_TRIG;
	rtrig_clear_done: R_TRIG;
	fb_ton_stow: TON;
	
	fb_rtrig_stow_deactivate1: R_TRIG;
	fb_rtrig_stow_deactivate: R_TRIG;
	b_execute_goto_Az: BOOL;
	R_TRIG_0: R_TRIG;
	R_TRIG_1: R_TRIG;
	rtrig_stop_goto_el: R_TRIG;
	rtrig_stop_goto_az: R_TRIG;
	fb_TON_2: TON;
	fb_TON_1: TON;
	r_goto_Az_rel: REAL;
	r_goto_El_rel: LREAL;
	r_goto_fi_rel: LREAL;
	fb_ton_stow1: TON;
	rtrig_reset_stop_el: R_TRIG;
	rtrig_reset_stop_Fi: R_TRIG;
END_VAR
VAR // added by the converter: edge detectors and wires of the graphical bodies
    _w1, _w2 : BOOL;
END_VAR

(* CASE  CommandArbiter.Status.DscCmdAuthority OF
	DscCmdAuthorityType.EGUI: 
		 b_track_start:=FALSE;
		 b_start_goto_el:=FALSE;
	DscCmdAuthorityType.LMC:
		b_scc_goto:=FALSE;
	DscCmdAuthorityType.HHP:
		 b_track_start:=FALSE;
		 b_start_goto_el:=FALSE;
		b_scc_goto:=FALSE;
		b_track_on:=FALSE;
	DscCmdAuthorityType.NoAuthority:
		 b_track_start:=FALSE;
		 b_start_goto_el:=FALSE;
		b_scc_goto:=FALSE;
		b_track_on:=FALSE; 
 END_CASE

*)

IF CommandArbiter.Status.DscCmdAuthority = 3 THEN
	 b_EGUI_control:=1;
	 b_LMC_control:=0;
	 b_HHP_control:=0;
ELSIF  CommandArbiter.Status.DscCmdAuthority = 1 THEN
	 b_EGUI_control:=0;
	 b_LMC_control:=1;
	 b_HHP_control:=0;
ELSIF CommandArbiter.Status.DscCmdAuthority = 2 THEN
	 b_EGUI_control:=0;
	 b_LMC_control:=0;
	 b_HHP_control:=1;
	 b_enable_az_1:=FALSE;
	 b_enable_az_2:=FALSE;
	 b_enable_el_3:=FALSE;
ELSE
	b_EGUI_control:=0;
	 b_LMC_control:=0;
	 b_HHP_control:=0;	 
END_IF

(***********Management.DscState***********)
IF azimuth.Status.AxisState=axisstatetype.StartUp OR elevation.Status.AxisState=axisstatetype.StartUp THEN
	Management.Status.DscState:=DscstateType.StartUp;
END_IF

IF azimuth.Status.AxisState=axisstatetype.Standby AND elevation.Status.AxisState=axisstatetype.Standby THEN
	Management.Status.DscState:=DscstateType.Standby;
END_IF

IF azimuth.Status.AxisState=axisstatetype.Activating OR elevation.Status.AxisState=axisstatetype.Activating THEN
	Management.Status.DscState:=DscstateType.Activating;
END_IF

IF azimuth.Status.AxisState=axisstatetype.Deactivating OR elevation.Status.AxisState=axisstatetype.Deactivating THEN
	Management.Status.DscState:=DscstateType.Deactivating;
END_IF

IF azimuth.Status.AxisState=axisstatetype.Standstill OR elevation.Status.AxisState=axisstatetype.Standstill THEN
	Management.Status.DscState:=DscstateType.Standstill;
END_IF

IF azimuth.Status.AxisState=axisstatetype.Stopping OR elevation.Status.AxisState=axisstatetype.Stopping THEN
	Management.Status.DscState:=DscstateType.stopping;
END_IF

IF azimuth.Status.AxisState=axisstatetype.Jog OR elevation.Status.AxisState=axisstatetype.Jog THEN
	Management.Status.DscState:=DscstateType.Jog;
END_IF

IF azimuth.Status.AxisState=axisstatetype.Slew OR elevation.Status.AxisState=axisstatetype.Slew THEN //capitalise S in slew
	Management.Status.DscState:=DscstateType.slew;
END_IF

IF azimuth.Status.AxisState=axisstatetype.Track AND elevation.Status.AxisState=axisstatetype.Track THEN
	Management.Status.DscState:=DscstateType.Track;
END_IF

IF azimuth.Status.AxisState=axisstatetype.Stowed THEN
	Management.Status.DscState:=DscstateType.Stowed;
	b_start_goto_Az:=FALSE;	
	b_start_goto_El:=FALSE;
	b_clear_err_Az:=FALSE;
	b_clear_err_El:=FALSE;
	b_clear_err_Fi:=FALSE;
	b_clear_err:=FALSE;
END_IF
IF azimuth.Status.AxisState=axisstatetype.Locked OR elevation.Status.AxisState=axisstatetype.Locked THEN
	Management.Status.DscState:=DscstateType.Locked;
	b_start_goto_Az:=FALSE;	
	b_start_goto_El:=FALSE;
	b_clear_err_Az:=FALSE;
	b_clear_err_El:=FALSE;
	b_clear_err_Fi:=FALSE;
	b_clear_err:=FALSE;
END_IF

IF azimuth.Status.AxisState=axisstatetype.Locked_Stowed OR elevation.Status.AxisState=axisstatetype.Locked_Stowed THEN
	Management.Status.DscState:=DscstateType.Locked_Stowed;
	b_start_goto_Az:=FALSE;	
	b_start_goto_El:=FALSE;
	b_clear_err_Az:=FALSE;
	b_clear_err_El:=FALSE;
	b_clear_err_Fi:=FALSE;
	b_clear_err:=FALSE;
END_IF

// This one isn't going to work 
IF b_stow_pin_limit_lock AND (azimuth.Status.AxisState=axisstatetype.Locked OR elevation.Status.AxisState=axisstatetype.Locked) THEN     // Need to check Errors and interlocks to go into locked
	Management.Status.DscState:=DscstateType.Locked_Stowed;
END_IF

(*IF b_in_Estop THEN
	Management.Status.DscState:=DscstateType.Locked;  //Axis also need to go into locked state
END_IF
*)


// Work out where FiPOS is 
IF b_goto_done_Fi THEN 
	IF r_pos_fi_v < gc_r_band_optical+gc_r_band_tolerance AND r_pos_fi_v > gc_r_band_optical-gc_r_band_tolerance THEN 
		Management.Status.FiPos:= bandtype.Optical;
	ELSIF
		r_pos_fi_v < gc_r_band_1+gc_r_band_tolerance AND r_pos_fi_v > gc_r_band_1-gc_r_band_tolerance THEN 
		Management.Status.FiPos:= bandtype.Band_1;
	ELSIF
		r_pos_fi_v < gc_r_band_2+gc_r_band_tolerance AND r_pos_fi_v > gc_r_band_2-gc_r_band_tolerance THEN 
		Management.Status.FiPos:= bandtype.Band_2;
	ELSIF
		r_pos_fi_v < gc_r_band_3+gc_r_band_tolerance AND r_pos_fi_v > gc_r_band_3-gc_r_band_tolerance THEN 
		Management.Status.FiPos:= bandtype.Band_3;
	ELSIF
		r_pos_fi_v < gc_r_band_4+gc_r_band_tolerance AND r_pos_fi_v > gc_r_band_4-gc_r_band_tolerance THEN 
		Management.Status.FiPos:= bandtype.Band_4;
	ELSIF
		r_pos_fi_v < gc_r_band_5a+gc_r_band_tolerance AND r_pos_fi_v > gc_r_band_5a-gc_r_band_tolerance THEN 
		Management.Status.FiPos:= bandtype.Band_5a;
	ELSIF
		r_pos_fi_v < gc_r_band_5b+gc_r_band_tolerance AND r_pos_fi_v > gc_r_band_5b-gc_r_band_tolerance THEN 
		Management.Status.FiPos:= bandtype.Band_5b;
	ELSIF
		r_pos_fi_v < gc_r_band_6+gc_r_band_tolerance AND r_pos_fi_v > gc_r_band_6-gc_r_band_tolerance THEN 
		Management.Status.FiPos:= bandtype.Band_6;
	ELSE
		Management.Status.FiPos:= bandtype.Unknown;
	END_IF

END_IF


//Management.Status.FiPos:=Current_FIPos; // this needs to be of band type 
Management.Status.HHP_Cncted:=b_HHP_Connected;
Management.Status.HHP_Az:=b_HHP_AZ;
Management.Status.HHP_El:=b_HHP_EL;
IF b_HHP_AZ = FALSE AND b_HHP_EL= FALSE THEN
	Management.Status.HHP_Fi:=TRUE;
ELSE
	Management.Status.HHP_Fi:=FALSE;
END_IF
IF b_HHP_move_cw_slow OR b_HHP_move_cw_fast THEN
	Management.Status.HHP_Dir_Plus	:= TRUE;
ELSE
	Management.Status.HHP_Dir_Plus	:= FALSE;
END_IF
IF b_HHP_move_ccw_slow OR b_HHP_move_ccw_fast THEN
	Management.Status.HHP_Dir_Minus:= TRUE;
ELSE
	Management.Status.HHP_Dir_Minus:= FALSE;
END_IF

(*********NamePlate**********)
Management.NamePlate.RunHours:=r_operation_hour;

count_i:=count_i+1;
IF count_i = 5 THEN
	R_total_distance_AZ:=ABS(r_pos_az-R_total_distance_AZ_old)+R_total_distance_AZ;
	R_total_distance_AZ_old:=r_pos_az;
	R_total_distance_EL_deg:=ABS(r_pos_el-R_total_distance_el_deg_old)+R_total_distance_el_deg;
	R_total_distance_EL_m:=R_total_distance_EL_deg/K_gear_ratio;
	R_total_distance_el_deg_old:=r_pos_el;
	R_total_distance_FI:=ABS(r_pos_FI-R_total_distance_FI_old)+R_total_distance_FI;
	R_total_distance_FI_old:=r_pos_FI;
	count_i:=0;
END_IF

Management.NamePlate.TotalDist_Az:=R_total_distance_AZ;
Management.NamePlate.TotalDist_El_deg:=R_total_distance_EL_deg;
Management.NamePlate.TotalDist_El_m:=R_total_distance_EL_m;
Management.NamePlate.TotalDist_Fi:=R_total_distance_FI;

(*********TempHumidStatus**********)
Management.TempHumidStatus.HumidDriveCab:=LREAL_TO_REAL(HumidDriveCab);
Management.TempHumidStatus.TempDriveCab:=LREAL_TO_REAL(TempDriveCab);
Management.TempHumidStatus.HumidPSC_Inlet:=LREAL_TO_REAL(HumidPSC_Inlet);
Management.TempHumidStatus.TempPSC_Inlet:=LREAL_TO_REAL(TempPSC_Inlet);
Management.TempHumidStatus.HumidPSC_Outlet:=LREAL_TO_REAL(HumidPSC_Outlet);
Management.TempHumidStatus.TempPSC_Outlet:=LREAL_TO_REAL(TempPSC_Outlet);
Management.TempHumidStatus.TempEMISC_Outlet:=LREAL_TO_REAL(TempEMISC_Outlet);

(*********PowerStatus**********)
Management.PowerStatus.SpdFnctnl_PDU1:=b_MAIN_PD_SPD_on;
Management.PowerStatus.SpdFnctnl_PDU2:=b_PSC_PD_SPD_on;
Management.PowerStatus.cbEMISC:=b_PSC_PD_EMISC_Breaker_on;
Management.PowerStatus.cbFan_PSC:=b_PSC_PD_FAN_Breaker_on;
Management.PowerStatus.cbPSC_Spare:=b_PSC_PD_spare;
Management.PowerStatus.cbHe_Comp:=b_MAIN_PD_Compressor_breaker_on;
Management.PowerStatus.cbPDU_Fi:=b_MAIN_PD_FI_Breaker_on;
Management.PowerStatus.cbPED_Spare:=b_MAIN_PD_spare;
Management.PowerStatus.ActPwrCnsm:= ApparentPowerConsumption; // Needs to be updated with real number
Management.PowerStatus.CurrentPh1:= LREAL_TO_REAL(CurrentPh1);
Management.PowerStatus.CurrentPh2:=LREAL_TO_REAL(CurrentPh2);
Management.PowerStatus.CurrentPh3:=LREAL_TO_REAL(CurrentPh3);
Management.PowerStatus.FrequencyPh1:=LREAL_TO_REAL(FrequencyPh1);
Management.PowerStatus.FrequencyPh2:=LREAL_TO_REAL(FrequencyPh2);
Management.PowerStatus.FrequencyPh3:=LREAL_TO_REAL(FrequencyPh3);
Management.PowerStatus.VoltagePh1:=LREAL_TO_REAL(VoltagePh1);
Management.PowerStatus.VoltagePh2:=LREAL_TO_REAL(VoltagePh2);
Management.PowerStatus.VoltagePh3:=LREAL_TO_REAL(VoltagePh3);
Management.PowerStatus.PowerFactor:=LREAL_TO_REAL(PowerFactor);

//Management.PowerStatus.LowPowerActive:=0;  

(*********ErrorStatus**********)

//Management.ErrorStatus.errAuthLost:=0;
Management.ErrorStatus.errAzimuth:=(axisdata[1].Axis_Error OR axisdata[2].Axis_Error);  
Management.ErrorStatus.errElevation:=(axisdata[3].Axis_Error);  
Management.ErrorStatus.errFeedindexer:=(axisdata[4].Axis_Error OR axisdata[5].Axis_Error); 
Management.ErrorStatus.errPoint:=0;
IF safety.Status.SafetyState=0 THEN
	Management.ErrorStatus.errSafety:=0;
ELSE
	Management.ErrorStatus.errSafety:=1;
END_IF
Management.ErrorStatus.errTime:=axisdata[10].Axis_Error;
Management.ErrorStatus.errCmd:=Command_Arbiter_error;
Management.ErrorStatus.errTrack:=(NOT(tracking.Status.tr_initOk) AND b_track_on);
Management.ErrorStatus.errStwPin:=NOT((b_stow_pin_limit_lock XOR NOT(b_stow_pin_limit_unlock))XOR(b_stow_pin_retract XOR b_stow_pin_deploy));
IF status_code1 = 'F8070' OR status_code2 = 'F8070' OR status_code3 = 'F8070' OR status_code4 = 'F8070' OR status_code5 = 'F8070' THEN
	Management.ErrorStatus.errPwr24VDC:=1;
ELSE
	Management.ErrorStatus.errPwr24VDC:=0;
END_IF
IF status_code1 = 'F2802' OR status_code2 = 'F2802' OR status_code3 = 'F2802' OR status_code4 = 'F2802' OR status_code5 = 'F2802' THEN
	Management.ErrorStatus.errPwr400VAC:=1;
ELSE
	Management.ErrorStatus.errPwr400VAC:=0;
END_IF
IF status_code1 = 'F2802' OR status_code2 = 'F2802' OR status_code3 = 'F2802' OR status_code4 = 'F2802' OR status_code5 = 'F2802' THEN
	Management.ErrorStatus.errPwr400VAC:=1;
ELSE
	Management.ErrorStatus.errPwr400VAC:=0;
END_IF
IF status_code1 = 'F8091' OR status_code2 = 'F8091' OR status_code3 = 'F8091' OR status_code4 = 'F8091' OR status_code5 = 'F8091' THEN
	Management.ErrorStatus.errPwr400VAC:=1;
ELSE
	Management.ErrorStatus.errPwr400VAC:=0;
END_IF
//	Management.ErrorStatus.errPwrMeterComms:=0;
//	Management.ErrorStatus.errTiltOneComms:=0;
//	Management.ErrorStatus.errTiltOneIoUnit:=0;
//	Management.ErrorStatus.errTiltTwoComms:=0;
//	Management.ErrorStatus.errTiltTwoIoUnit:=0;

Management.ErrorStatus.errGeneral:=(Management.ErrorStatus.errAzimuth OR Management.ErrorStatus.errElevation OR Management.ErrorStatus.errFeedindexer OR Management.ErrorStatus.errSafety OR Management.ErrorStatus.errTime OR Management.ErrorStatus.errTrack OR Management.ErrorStatus.errPoint);
Management.ErrorStatus.errMngmnt:=Management.ErrorStatus.errGeneral;

(*********WarningStatus**********)
//IF gc_b_sim_on = 0 THEN 
	Management.WarningStatus.waAzimuth:=(axisdata[1].Axis_Warning OR axisdata[2].Axis_Warning);
    Management.WarningStatus.waElevation:=(axisdata[3].Axis_Warning);
    Management.WarningStatus.waFeedindexer:=(axisdata[4].Axis_Warning OR axisdata[5].Axis_Warning);
//ELSIF gc_b_sim_on =1 THEN
//	Management.WarningStatus.waAzimuth:=(

Management.WarningStatus.waCmd:=0;
Management.WarningStatus.waPoint:=0;
Management.WarningStatus.waSafety:=0;
Management.WarningStatus.waStwPin:=0;
Management.WarningStatus.waPoint:=0;
Management.WarningStatus.waTime:=0;
Management.WarningStatus.waTrack:=0;
Management.WarningStatus.waDoorDrive:=b_DriveCabinetDoor_Estop;
Management.WarningStatus.waDoorEMISC:=b_EMISCDoor_Estop;
Management.WarningStatus.waDoorPED:=b_DSDoor_Estop;
Management.WarningStatus.waDoorPSC:=b_PSCDoor_Estop;
Management.WarningStatus.waHatchPscRoof:=0;
Management.WarningStatus.waHatchAzBearing:=b_AZ_Hatch;
Management.WarningStatus.waHornOn:=b_Horn;
//Management.WarningStatus.waOverTempDrive
//Management.WarningStatus.waOverTempEMISC
//Management.WarningStatus.waDoorPED
//Management.WarningStatus.waDoorPSC
Management.WarningStatus.waSafe2ApproachLight:=0;

// Power mode control 
// Need to limit velocity and acceleration to keep the power below the limit 


// Run Ladder logic
P_Opcua_Management.A_CLR_ERR();
P_Opcua_Management.A_STOP();
P_Opcua_Management.A_GOTO();

ACTION A_STOP:
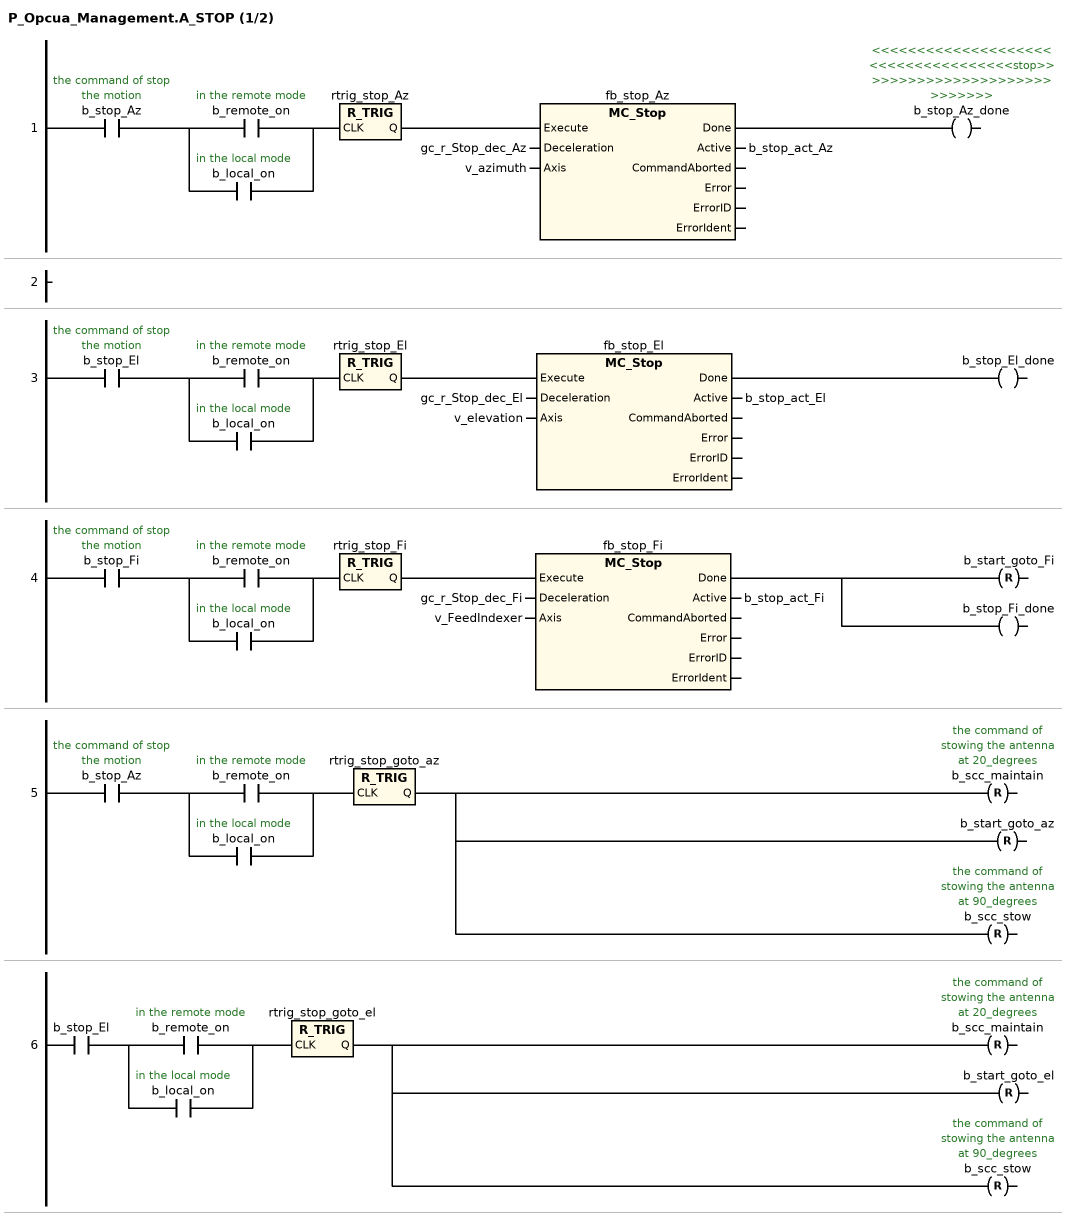
// NETWORK 1
//   b_stop_Az: the command of stop the motion
//   b_remote_on: in the remote mode
//   b_local_on: in the local mode
//   v_azimuth: Virtual axis "v_azimuth" with axis number 7
//   b_stop_Az_done: <<<<<<<<<<<<<<<<<<<<<<<<<<<<<<<<<<<<stop>>>>>>>>>>>>>>>>>>>>>>>>>>>>>
rtrig_stop_Az(CLK := b_stop_Az AND (b_remote_on OR b_local_on)); // R_TRIG
fb_stop_Az(
    Execute := rtrig_stop_Az.Q,
    Deceleration := gc_r_Stop_dec_Az,
    Axis := v_azimuth,
    Active => b_stop_act_Az); // MC_Stop
b_stop_Az_done := fb_stop_Az.Done;

// NETWORK 2

// NETWORK 3
//   b_stop_El: the command of stop the motion
//   b_remote_on: in the remote mode
//   b_local_on: in the local mode
//   v_elevation: Virtual axis "v_elevation" with axis number 8
rtrig_stop_El(CLK := b_stop_El AND (b_remote_on OR b_local_on)); // R_TRIG
fb_stop_El(
    Execute := rtrig_stop_El.Q,
    Deceleration := gc_r_Stop_dec_El,
    Axis := v_elevation,
    Active => b_stop_act_El); // MC_Stop
b_stop_El_done := fb_stop_El.Done;

// NETWORK 4
//   b_stop_Fi: the command of stop the motion
//   b_remote_on: in the remote mode
//   b_local_on: in the local mode
//   v_FeedIndexer: Virtual axis "v_polarization" with axis number 9
rtrig_stop_Fi(CLK := b_stop_Fi AND (b_remote_on OR b_local_on)); // R_TRIG
fb_stop_Fi(
    Execute := rtrig_stop_Fi.Q,
    Deceleration := gc_r_Stop_dec_Fi,
    Axis := v_FeedIndexer,
    Active => b_stop_act_Fi); // MC_Stop
b_start_goto_Fi R= fb_stop_Fi.Done;
b_stop_Fi_done := fb_stop_Fi.Done;

// NETWORK 5
//   b_stop_Az: the command of stop the motion
//   b_remote_on: in the remote mode
//   b_local_on: in the local mode
//   b_scc_maintain: the command of stowing the antenna at 20_degrees
//   b_scc_stow: the command of stowing the antenna at 90_degrees
rtrig_stop_goto_az(CLK := b_stop_Az AND (b_remote_on OR b_local_on)); // R_TRIG
b_scc_maintain R= rtrig_stop_goto_az.Q;
b_start_goto_az R= rtrig_stop_goto_az.Q;
b_scc_stow R= rtrig_stop_goto_az.Q;

// NETWORK 6
//   b_remote_on: in the remote mode
//   b_local_on: in the local mode
//   b_scc_maintain: the command of stowing the antenna at 20_degrees
//   b_scc_stow: the command of stowing the antenna at 90_degrees
rtrig_stop_goto_el(CLK := b_stop_El AND (b_remote_on OR b_local_on)); // R_TRIG
b_scc_maintain R= rtrig_stop_goto_el.Q;
b_start_goto_el R= rtrig_stop_goto_el.Q;
b_scc_stow R= rtrig_stop_goto_el.Q;

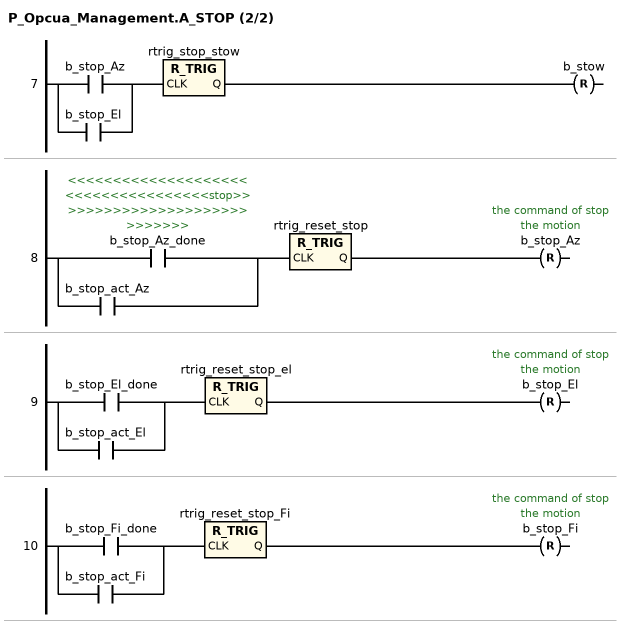
// NETWORK 7
rtrig_stop_stow(CLK := b_stop_Az OR b_stop_El); // R_TRIG
b_stow R= rtrig_stop_stow.Q;

// NETWORK 8
//   b_stop_Az_done: <<<<<<<<<<<<<<<<<<<<<<<<<<<<<<<<<<<<stop>>>>>>>>>>>>>>>>>>>>>>>>>>>>>
//   b_stop_Az: the command of stop the motion
rtrig_reset_stop(CLK := b_stop_Az_done OR b_stop_act_Az); // R_TRIG
b_stop_Az R= rtrig_reset_stop.Q;

// NETWORK 9
//   b_stop_El: the command of stop the motion
rtrig_reset_stop_el(CLK := b_stop_El_done OR b_stop_act_El); // R_TRIG
b_stop_El R= rtrig_reset_stop_el.Q;

// NETWORK 10
//   b_stop_Fi: the command of stop the motion
rtrig_reset_stop_Fi(CLK := b_stop_Fi_done OR b_stop_act_Fi); // R_TRIG
b_stop_Fi R= rtrig_reset_stop_Fi.Q;
END_ACTION

ACTION A_GOTO:
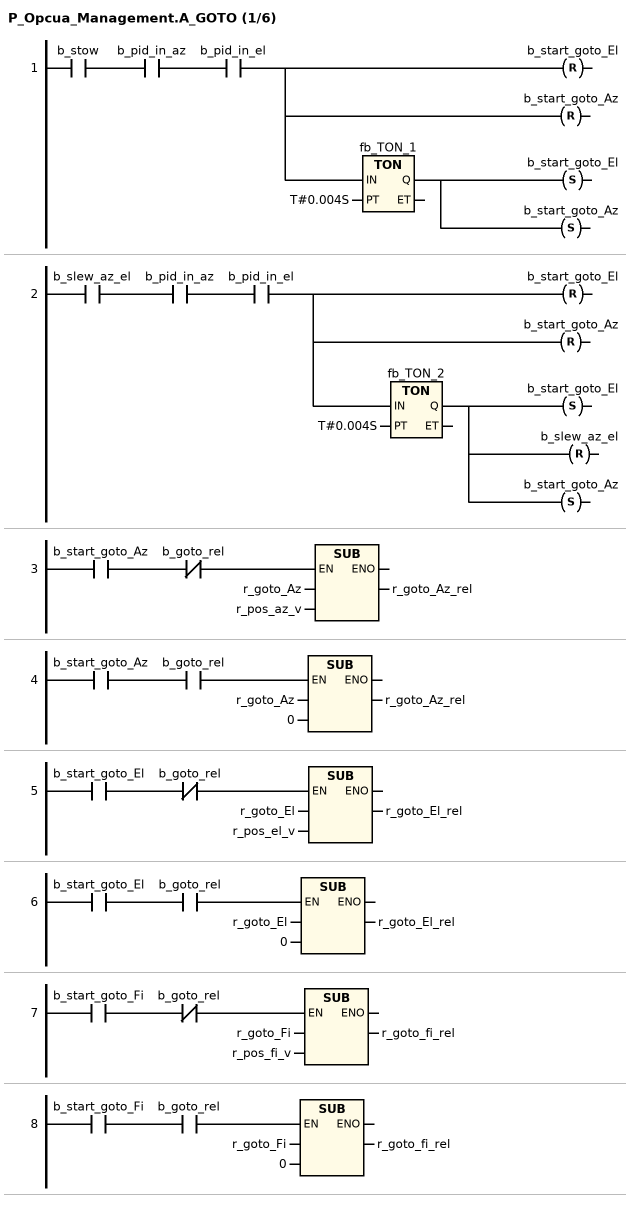
// NETWORK 1
_w1 := b_stow AND b_pid_in_az AND b_pid_in_el;
b_start_goto_El R= _w1;
b_start_goto_Az R= _w1;
fb_TON_1(IN := _w1, PT := T#0.004S); // TON
b_start_goto_El S= fb_TON_1.Q;
b_start_goto_Az S= fb_TON_1.Q;

// NETWORK 2
_w2 := b_slew_az_el AND b_pid_in_az AND b_pid_in_el;
b_start_goto_El R= _w2;
b_start_goto_Az R= _w2;
fb_TON_2(IN := _w2, PT := T#0.004S); // TON
b_start_goto_El S= fb_TON_2.Q;
b_slew_az_el R= fb_TON_2.Q;
b_start_goto_Az S= fb_TON_2.Q;

// NETWORK 3
IF b_start_goto_Az AND NOT b_goto_rel THEN r_goto_Az_rel := r_goto_Az - r_pos_az_v; END_IF

// NETWORK 4
IF b_start_goto_Az AND b_goto_rel THEN r_goto_Az_rel := r_goto_Az - 0; END_IF

// NETWORK 5
IF b_start_goto_El AND NOT b_goto_rel THEN r_goto_El_rel := r_goto_El - r_pos_el_v; END_IF

// NETWORK 6
IF b_start_goto_El AND b_goto_rel THEN r_goto_El_rel := r_goto_El - 0; END_IF

// NETWORK 7
IF b_start_goto_Fi AND NOT b_goto_rel THEN r_goto_fi_rel := r_goto_Fi - r_pos_fi_v; END_IF

// NETWORK 8
IF b_start_goto_Fi AND b_goto_rel THEN r_goto_fi_rel := r_goto_Fi - 0; END_IF

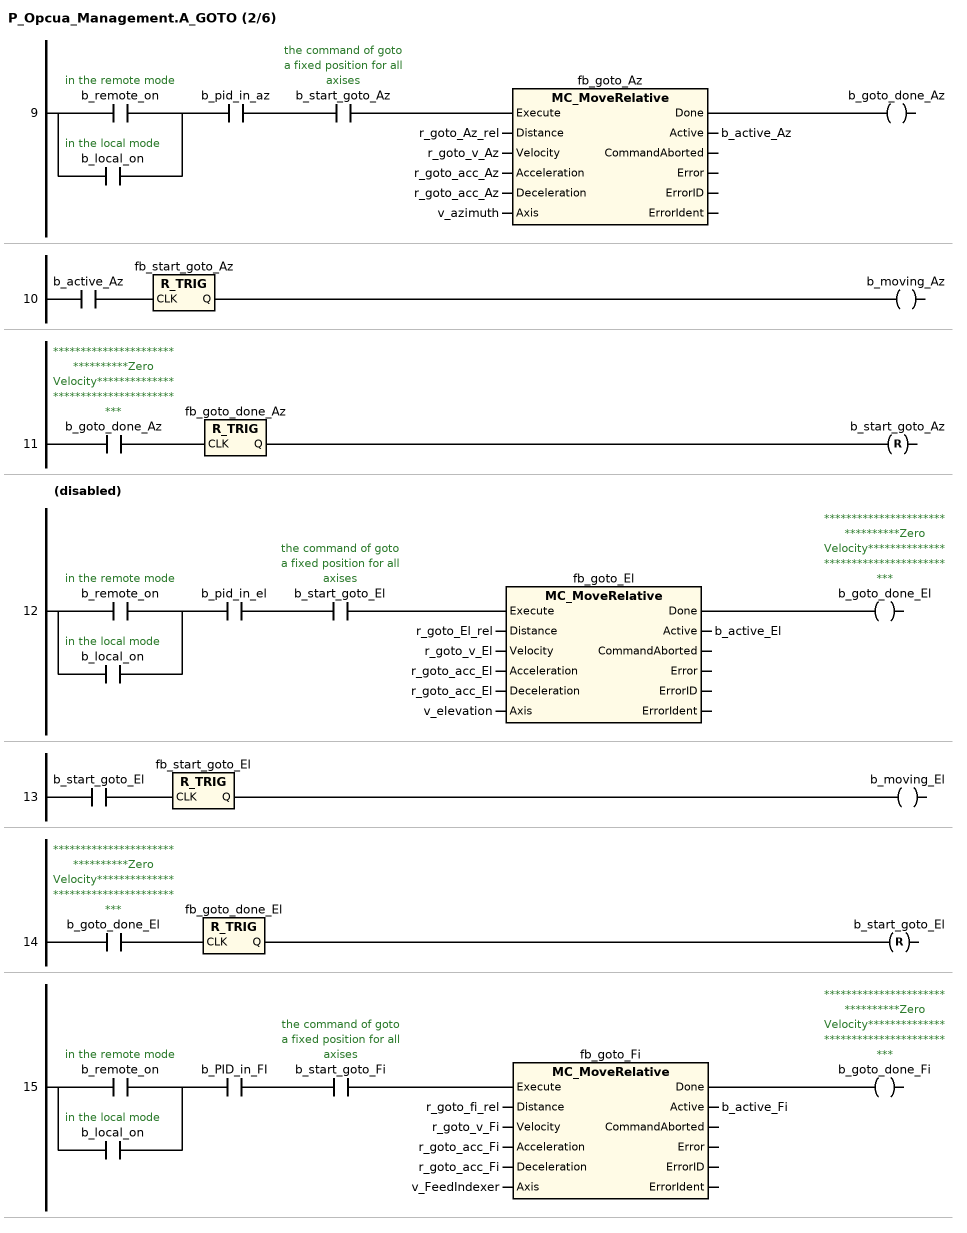
// NETWORK 9
//   b_remote_on: in the remote mode
//   b_local_on: in the local mode
//   b_start_goto_Az: the command of goto a fixed position for all axises
//   r_goto_Az_rel: actual value of goto
//   v_azimuth: Virtual axis "v_azimuth" with axis number 7
fb_goto_Az(
    Execute := (b_remote_on OR b_local_on) AND b_pid_in_az AND b_start_goto_Az,
    Distance := r_goto_Az_rel,
    Velocity := r_goto_v_Az,
    Acceleration := r_goto_acc_Az,
    Deceleration := r_goto_acc_Az,
    Axis := v_azimuth,
    Active => b_active_Az); // MC_MoveRelative
b_goto_done_Az := fb_goto_Az.Done;

// NETWORK 10
fb_start_goto_Az(CLK := b_active_Az); // R_TRIG
b_moving_Az := fb_start_goto_Az.Q;

// NETWORK 11
//   b_goto_done_Az: ********************************Zero Velocity***************************************
fb_goto_done_Az(CLK := b_goto_done_Az); // R_TRIG
b_start_goto_Az R= fb_goto_done_Az.Q;

// NETWORK 12 (disabled)
//   b_remote_on: in the remote mode
//   b_local_on: in the local mode
//   b_start_goto_El: the command of goto a fixed position for all axises
//   r_goto_El_rel: actual value of goto
//   v_elevation: Virtual axis "v_azimuth" with axis number 7
//   b_goto_done_El: ********************************Zero Velocity***************************************
// fb_goto_El(
//     Execute := (b_remote_on OR b_local_on) AND b_pid_in_el AND b_start_goto_El,
//     Distance := r_goto_El_rel,
//     Velocity := r_goto_v_El,
//     Acceleration := r_goto_acc_El,
//     Deceleration := r_goto_acc_El,
//     Axis := v_elevation,
//     Active => b_active_El); // MC_MoveRelative
// b_goto_done_El := fb_goto_El.Done;

// NETWORK 13
fb_start_goto_El(CLK := b_start_goto_El); // R_TRIG
b_moving_El := fb_start_goto_El.Q;

// NETWORK 14
//   b_goto_done_El: ********************************Zero Velocity***************************************
fb_goto_done_El(CLK := b_goto_done_El); // R_TRIG
b_start_goto_El R= fb_goto_done_El.Q;

// NETWORK 15
//   b_remote_on: in the remote mode
//   b_local_on: in the local mode
//   b_start_goto_Fi: the command of goto a fixed position for all axises
//   r_goto_fi_rel: actual value of goto
//   v_FeedIndexer: Virtual axis "v_azimuth" with axis number 7
//   b_goto_done_Fi: ********************************Zero Velocity***************************************
fb_goto_Fi(
    Execute := (b_remote_on OR b_local_on) AND b_PID_in_FI AND b_start_goto_Fi,
    Distance := r_goto_fi_rel,
    Velocity := r_goto_v_Fi,
    Acceleration := r_goto_acc_Fi,
    Deceleration := r_goto_acc_Fi,
    Axis := v_FeedIndexer,
    Active => b_active_Fi); // MC_MoveRelative
b_goto_done_Fi := fb_goto_Fi.Done;

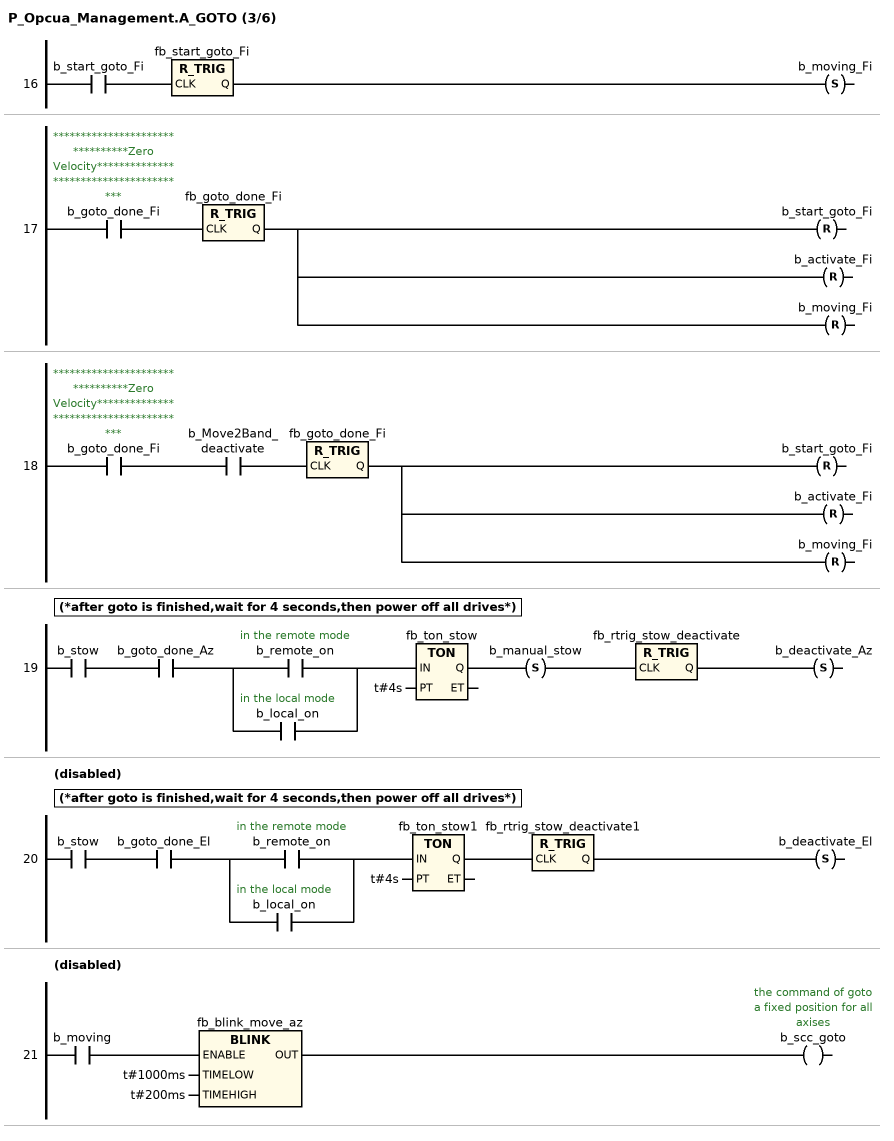
// NETWORK 16
fb_start_goto_Fi(CLK := b_start_goto_Fi); // R_TRIG
b_moving_Fi S= fb_start_goto_Fi.Q;

// NETWORK 17
//   b_goto_done_Fi: ********************************Zero Velocity***************************************
fb_goto_done_Fi(CLK := b_goto_done_Fi); // R_TRIG
b_start_goto_Fi R= fb_goto_done_Fi.Q;
b_activate_Fi R= fb_goto_done_Fi.Q;
b_moving_Fi R= fb_goto_done_Fi.Q;

// NETWORK 18
//   b_goto_done_Fi: ********************************Zero Velocity***************************************
fb_goto_done_Fi(CLK := b_goto_done_Fi AND b_Move2Band_deactivate); // R_TRIG
b_start_goto_Fi R= fb_goto_done_Fi.Q;
b_activate_Fi R= fb_goto_done_Fi.Q;
b_moving_Fi R= fb_goto_done_Fi.Q;

// NETWORK 19
//   fb_rtrig_stow_deactivate: the definition of rise trigger,The function block R_TRIG detects a rising edge.
//   fb_ton_stow: The function block Timer On Delay implements a turn-on delay
//   b_remote_on: in the remote mode
//   b_local_on: in the local mode
// label: (*after goto is finished,wait for 4 seconds,then power off all drives*)
fb_ton_stow(IN := b_stow AND b_goto_done_Az AND (b_remote_on OR b_local_on), PT := t#4s); // TON
b_manual_stow S= fb_ton_stow.Q;
fb_rtrig_stow_deactivate(CLK := fb_ton_stow.Q); // R_TRIG
b_deactivate_Az S= fb_rtrig_stow_deactivate.Q;

// NETWORK 20 (disabled)
//   fb_rtrig_stow_deactivate1: the definition of rise trigger,The function block R_TRIG detects a rising edge.
//   fb_ton_stow1: The function block Timer On Delay implements a turn-on delay
//   b_remote_on: in the remote mode
//   b_local_on: in the local mode
// label: (*after goto is finished,wait for 4 seconds,then power off all drives*)
// fb_ton_stow1(IN := b_stow AND b_goto_done_El AND (b_remote_on OR b_local_on), PT := t#4s); // TON
// fb_rtrig_stow_deactivate1(CLK := fb_ton_stow1.Q); // R_TRIG
// b_deactivate_El S= fb_rtrig_stow_deactivate1.Q;

// NETWORK 21 (disabled)
//   b_scc_goto: the command of goto a fixed position for all axises
// fb_blink_move_az(ENABLE := b_moving, TIMELOW := t#1000ms, TIMEHIGH := t#200ms); // BLINK
// b_scc_goto := fb_blink_move_az.OUT;

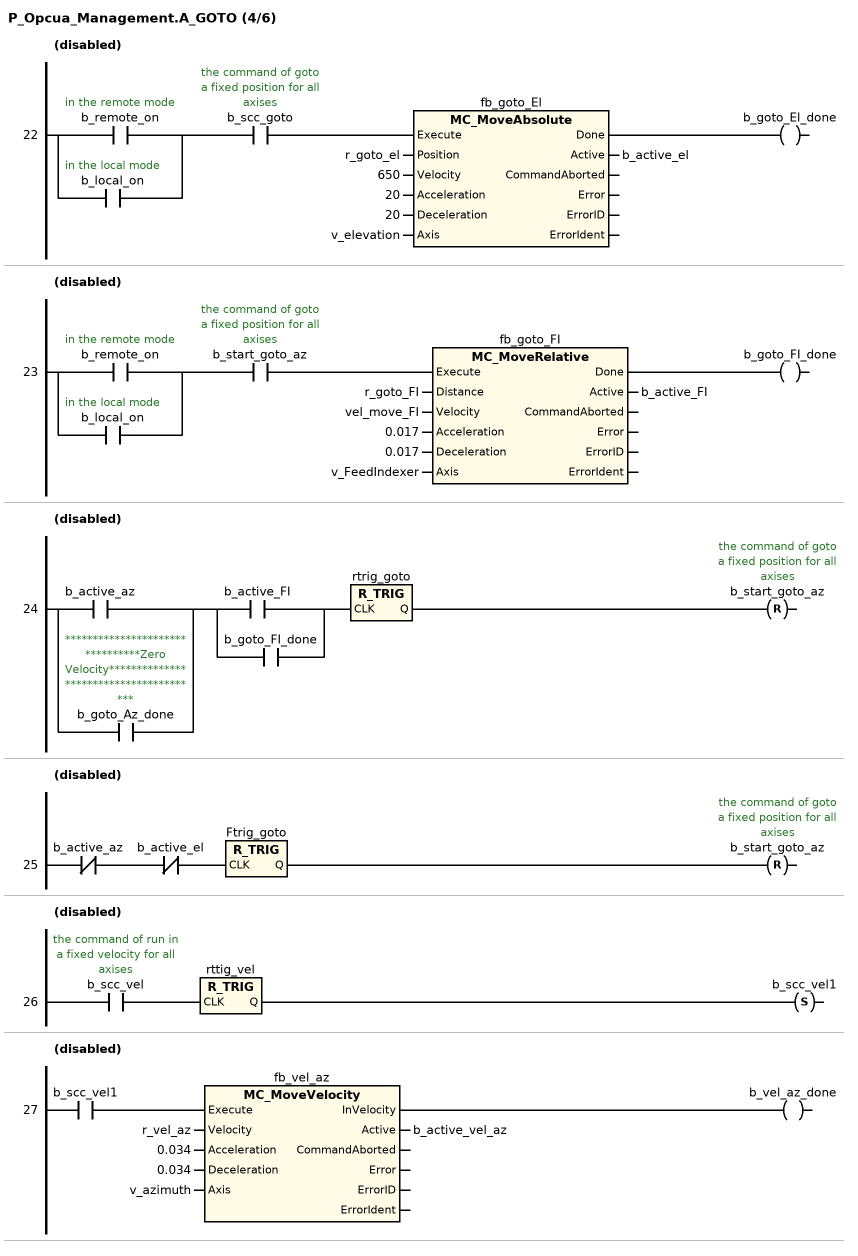
// NETWORK 22 (disabled)
//   b_remote_on: in the remote mode
//   b_local_on: in the local mode
//   b_scc_goto: the command of goto a fixed position for all axises
//   v_elevation: Virtual axis "v_elevation" with axis number 8
// fb_goto_El(
//     Execute := (b_remote_on OR b_local_on) AND b_scc_goto,
//     Position := r_goto_el,
//     Velocity := 650,
//     Acceleration := 20,
//     Deceleration := 20,
//     Axis := v_elevation,
//     Active => b_active_el); // MC_MoveAbsolute
// b_goto_El_done := fb_goto_El.Done;

// NETWORK 23 (disabled)
//   b_remote_on: in the remote mode
//   b_local_on: in the local mode
//   b_start_goto_az: the command of goto a fixed position for all axises
//   v_FeedIndexer: Virtual axis "v_polarization" with axis number 9
// fb_goto_FI(
//     Execute := (b_remote_on OR b_local_on) AND b_start_goto_az,
//     Distance := r_goto_FI,
//     Velocity := vel_move_FI,
//     Acceleration := 0.017,
//     Deceleration := 0.017,
//     Axis := v_FeedIndexer,
//     Active => b_active_FI); // MC_MoveRelative
// b_goto_FI_done := fb_goto_FI.Done;

// NETWORK 24 (disabled)
//   b_goto_Az_done: ********************************Zero Velocity***************************************
//   b_start_goto_az: the command of goto a fixed position for all axises
// rtrig_goto(CLK := (b_active_az OR b_goto_Az_done) AND (b_active_FI OR b_goto_FI_done)); // R_TRIG
// b_start_goto_az R= rtrig_goto.Q;

// NETWORK 25 (disabled)
//   b_start_goto_az: the command of goto a fixed position for all axises
// Ftrig_goto(CLK := NOT b_active_az AND NOT b_active_el); // R_TRIG
// b_start_goto_az R= Ftrig_goto.Q;

// NETWORK 26 (disabled)
//   b_scc_vel: the command of run in a fixed velocity for all axises
// rttig_vel(CLK := b_scc_vel); // R_TRIG
// b_scc_vel1 S= rttig_vel.Q;

// NETWORK 27 (disabled)
//   r_vel_az: ************vel*************
//   v_azimuth: Virtual axis "v_azimuth" with axis number 7
// fb_vel_az(
//     Execute := b_scc_vel1,
//     Velocity := r_vel_az,
//     Acceleration := 0.034,
//     Deceleration := 0.034,
//     Axis := v_azimuth,
//     Active => b_active_vel_az); // MC_MoveVelocity
// b_vel_az_done := fb_vel_az.InVelocity;

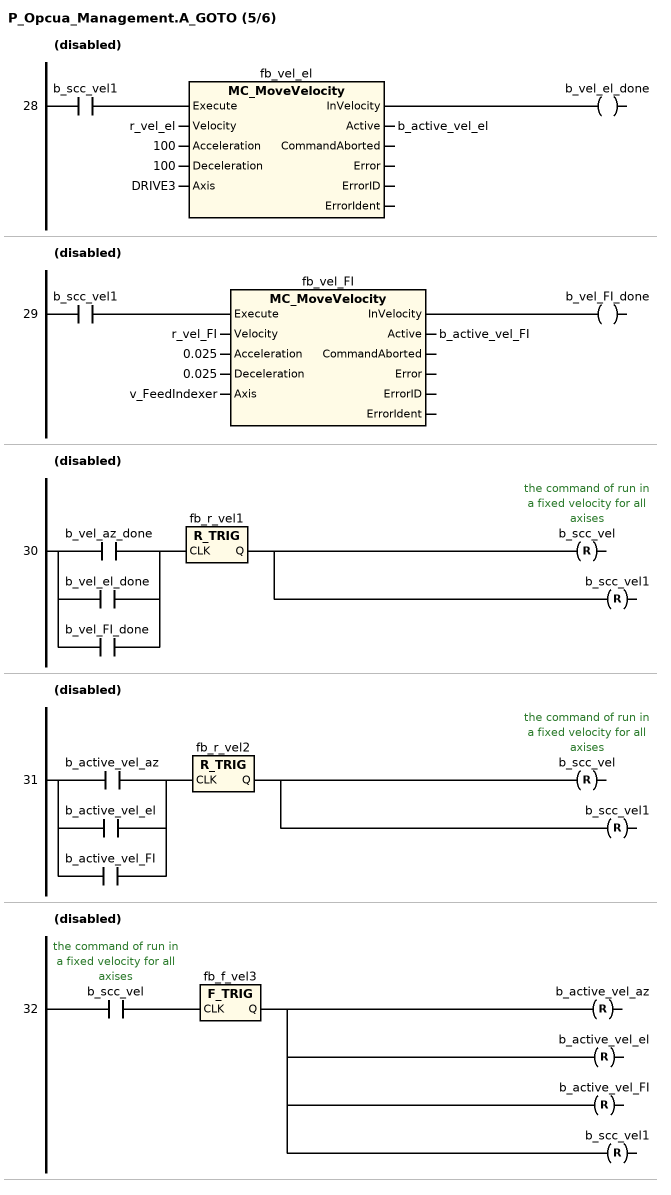
// NETWORK 28 (disabled)
//   DRIVE3: Virtual axis "v_elevation" with axis number 8
// fb_vel_el(
//     Execute := b_scc_vel1,
//     Velocity := r_vel_el,
//     Acceleration := 100,
//     Deceleration := 100,
//     Axis := DRIVE3,
//     Active => b_active_vel_el); // MC_MoveVelocity
// b_vel_el_done := fb_vel_el.InVelocity;

// NETWORK 29 (disabled)
//   v_FeedIndexer: Virtual axis "v_polarization" with axis number 9
// fb_vel_FI(
//     Execute := b_scc_vel1,
//     Velocity := r_vel_FI,
//     Acceleration := 0.025,
//     Deceleration := 0.025,
//     Axis := v_FeedIndexer,
//     Active => b_active_vel_FI); // MC_MoveVelocity
// b_vel_FI_done := fb_vel_FI.InVelocity;

// NETWORK 30 (disabled)
//   b_scc_vel: the command of run in a fixed velocity for all axises
// fb_r_vel1(CLK := b_vel_az_done OR b_vel_el_done OR b_vel_FI_done); // R_TRIG
// b_scc_vel R= fb_r_vel1.Q;
// b_scc_vel1 R= fb_r_vel1.Q;

// NETWORK 31 (disabled)
//   b_scc_vel: the command of run in a fixed velocity for all axises
// fb_r_vel2(CLK := b_active_vel_az OR b_active_vel_el OR b_active_vel_FI); // R_TRIG
// b_scc_vel R= fb_r_vel2.Q;
// b_scc_vel1 R= fb_r_vel2.Q;

// NETWORK 32 (disabled)
//   b_scc_vel: the command of run in a fixed velocity for all axises
// fb_f_vel3(CLK := b_scc_vel); // F_TRIG
// b_active_vel_az R= fb_f_vel3.Q;
// b_active_vel_el R= fb_f_vel3.Q;
// b_active_vel_FI R= fb_f_vel3.Q;
// b_scc_vel1 R= fb_f_vel3.Q;

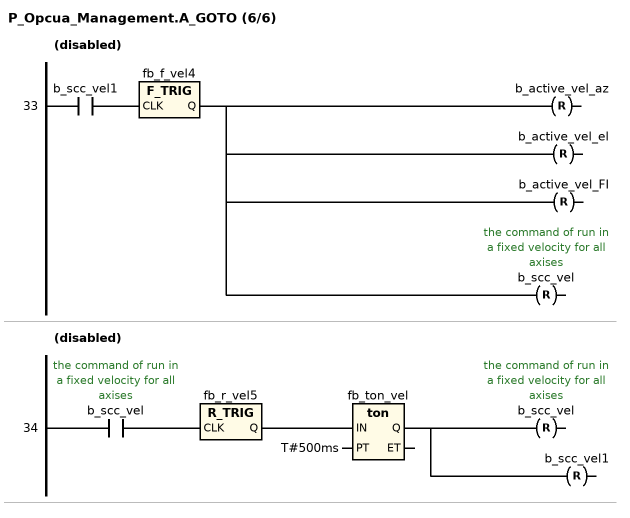
// NETWORK 33 (disabled)
//   b_scc_vel: the command of run in a fixed velocity for all axises
// fb_f_vel4(CLK := b_scc_vel1); // F_TRIG
// b_active_vel_az R= fb_f_vel4.Q;
// b_active_vel_el R= fb_f_vel4.Q;
// b_active_vel_FI R= fb_f_vel4.Q;
// b_scc_vel R= fb_f_vel4.Q;

// NETWORK 34 (disabled)
//   b_scc_vel: the command of run in a fixed velocity for all axises
// fb_r_vel5(CLK := b_scc_vel); // R_TRIG
// fb_ton_vel(IN := fb_r_vel5.Q, PT := T#500ms); // ton
// b_scc_vel R= fb_ton_vel.Q;
// b_scc_vel1 R= fb_ton_vel.Q;
END_ACTION

ACTION A_CLR_ERR:
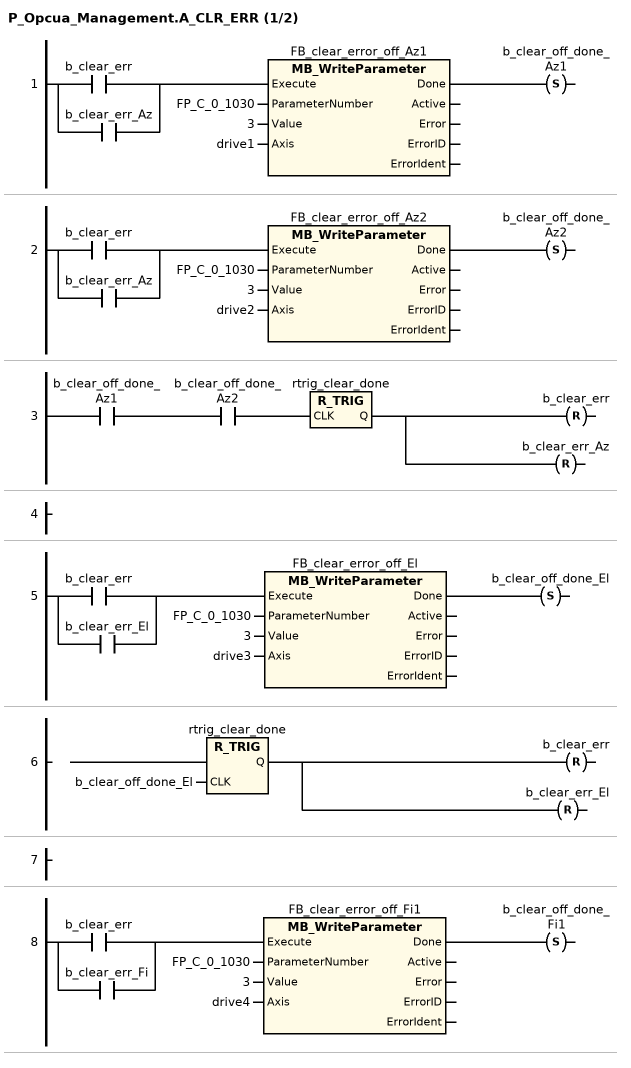
// NETWORK 1
//   FP_C_0_1030: Command: Clear all control errors
//   drive1: Real axis "Drive1" with axis number 1
FB_clear_error_off_Az1(
    Execute := b_clear_err OR b_clear_err_Az,
    ParameterNumber := FP_C_0_1030,
    Value := 3,
    Axis := drive1); // MB_WriteParameter
b_clear_off_done_Az1 S= FB_clear_error_off_Az1.Done;

// NETWORK 2
//   FP_C_0_1030: Command: Clear all control errors
//   drive2: Real axis "Drive1" with axis number 1
FB_clear_error_off_Az2(
    Execute := b_clear_err OR b_clear_err_Az,
    ParameterNumber := FP_C_0_1030,
    Value := 3,
    Axis := drive2); // MB_WriteParameter
b_clear_off_done_Az2 S= FB_clear_error_off_Az2.Done;

// NETWORK 3
rtrig_clear_done(CLK := b_clear_off_done_Az1 AND b_clear_off_done_Az2); // R_TRIG
b_clear_err R= rtrig_clear_done.Q;
b_clear_err_Az R= rtrig_clear_done.Q;

// NETWORK 4

// NETWORK 5
//   FP_C_0_1030: Command: Clear all control errors
//   drive3: Real axis "Drive1" with axis number 1
FB_clear_error_off_El(
    Execute := b_clear_err OR b_clear_err_El,
    ParameterNumber := FP_C_0_1030,
    Value := 3,
    Axis := drive3); // MB_WriteParameter
b_clear_off_done_El S= FB_clear_error_off_El.Done;

// NETWORK 6
rtrig_clear_done(CLK := b_clear_off_done_El); // R_TRIG
b_clear_err R= rtrig_clear_done.Q;
b_clear_err_El R= rtrig_clear_done.Q;

// NETWORK 7

// NETWORK 8
//   FP_C_0_1030: Command: Clear all control errors
//   drive4: Real axis "Drive1" with axis number 1
FB_clear_error_off_Fi1(
    Execute := b_clear_err OR b_clear_err_Fi,
    ParameterNumber := FP_C_0_1030,
    Value := 3,
    Axis := drive4); // MB_WriteParameter
b_clear_off_done_Fi1 S= FB_clear_error_off_Fi1.Done;

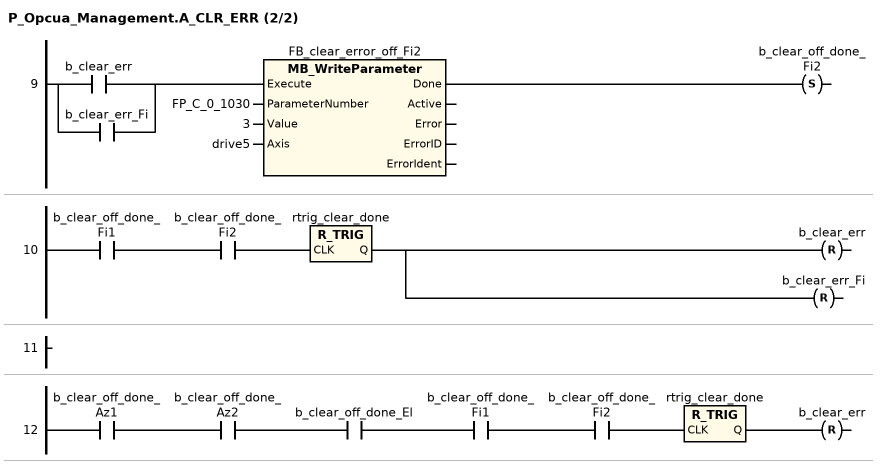
// NETWORK 9
//   FP_C_0_1030: Command: Clear all control errors
//   drive5: Real axis "Drive1" with axis number 1
FB_clear_error_off_Fi2(
    Execute := b_clear_err OR b_clear_err_Fi,
    ParameterNumber := FP_C_0_1030,
    Value := 3,
    Axis := drive5); // MB_WriteParameter
b_clear_off_done_Fi2 S= FB_clear_error_off_Fi2.Done;

// NETWORK 10
rtrig_clear_done(CLK := b_clear_off_done_Fi1 AND b_clear_off_done_Fi2); // R_TRIG
b_clear_err R= rtrig_clear_done.Q;
b_clear_err_Fi R= rtrig_clear_done.Q;

// NETWORK 11

// NETWORK 12
rtrig_clear_done(CLK := b_clear_off_done_Az1 AND b_clear_off_done_Az2 AND b_clear_off_done_El AND b_clear_off_done_Fi1 AND b_clear_off_done_Fi2); // R_TRIG
b_clear_err R= rtrig_clear_done.Q;
END_ACTION

END_PROGRAM

// IndraMotionMlc1/Application/POUs/OPCUA/OPCUA_Node/P_Opcua_Tracking
{attribute 'linkalways'}
PROGRAM P_Opcua_Tracking
VAR_INPUT
	
	i_length: UINT;
	tai: ARRAY [1..1000] OF LREAL;
	Az: ARRAY [1..1000] OF LREAL;
	El: ARRAY [1..1000] OF LREAL;
	
END_VAR

VAR
	index: UINT; // Index used for addressing points in the tracking data arrays. 
	
	IL_LowPass_OnSource: IL_StateVariableType01;
	b_test: BOOL;
	
END_VAR


// Switch track on if the starttime has been reached
IF b_track_start AND (lr_track_start_time <= Time_cds.Status.TAIoffset) THEN 
	b_track_on:=1;
	b_track_start:=0;
END_IF

//IF i_length>0 THEN  // Load table into stack 
	
	
//END_IF

// Calculate whether the dish is on source. 

IF b_track_on THEN 
	IF  tracking.status.OnSourceDev <= Tracking.Status.OnSourceThreshold THEN 
		Management.Status.OnSource:=1;
	ELSE
		Management.Status.OnSource:=0;	
	END_IF
ELSE
	Management.Status.OnSource:=0;
END_IF

//Tracking.Status.act_statOffset_value_El  Updated in P_Track_cubic
//Tracking.Status.act_statOffset_value_Xel Updated in P_Track_cubic
//Tracking.Status.OnSourceDev              Updated in P_Track_cubic
//Tracking.Status.OnSourceThreshold        Updated in SetOnSourceThreshold
//Tracking.Status.p_desired_Az;            Updated in P_Track_cubic
//Tracking.Status.p_desired_El;            Updated in P_Track_cubic
//Tracking.Status.ThresholdTimePeriod      Updated in SetOnSourceThreshold
IF Management.Status.DscState=DscStatetype.Standby OR Management.Status.DscState=DscStatetype.Standstill OR Management.Status.DscState=DscStatetype.Slew OR Management.Status.DscState=DscStatetype.Track THEN 
	Tracking.Status.tr_initOk:=1;
ELSE 
	Tracking.Status.tr_initOk:=0;
END_IF

Tracking.Status.tr_obj_valid:= Tracking.TableStatus.pts_DataValid;
Tracking.Status.tr_selPoly:= 0;

IF Tracking.TableStatus.pts_DataValid THEN
	Tracking.Status.tr_TimeRemaining:= ABS(track_table[i_End].TAIoffset - track_table[i_Start].TAIoffset);
ELSE
	Tracking.Status.tr_TimeRemaining:=0;
END_IF

IF (track_table[i_End].TAIoffset)>(Time_cds.Status.TAIoffset+600) THEN  // Minimum of 10min track data available . 
	Tracking.Status.tr_valid:=1;
ELSE
	Tracking.Status.tr_valid:=0;
END_IF

Tracking.TableStatus.act_pt_act_index := INT_TO_UINT(i_Start);
Tracking.TableStatus.act_pt_end_index := INT_TO_UINT(i_End);
Tracking.TableStatus.act_pt_value_Az:= track_table[i_Start].Azimuth;
Tracking.TableStatus.act_pt_value_El:= track_table[i_Start].Elevation;
//Tracking.TableStatus.LastLoadMode; Updated in TrackloadTable
IF i_num_stack_left > 10 THEN
	Tracking.TableStatus.pts_Completed:=0; 
	ELSE
	Tracking.TableStatus.pts_Completed:=1;
END_IF
IF Tracking.TableStatus.pts_Completed THEN 
	Tracking.TableStatus.pts_DataValid:=0; // Once a track is finnished then there is no valid data to trck with. 
END_IF
Tracking.TableStatus.pts_Err:=0; 
//Tracking.TableStatus.pts_Interpol;  Updated in Track Start
Tracking.TableStatus.pts_InterpolError:=0;  // Don't have code for detecting interpolaor errors yet
Tracking.TableStatus.pts_Running:=b_track_on;
Tracking.TableStatus.pts_StartPos:=b_track_on;

IF i_num_stack_left<=60 AND i_num_stack_left >= 70 THEN
	Tracking.TableStatus.pts_TableAlmostFull:=1;
ELSE 
	Tracking.TableStatus.pts_TableAlmostFull:=0;
END_IF

P_Opcua_Tracking.A_Utils();

ACTION A_Utils:
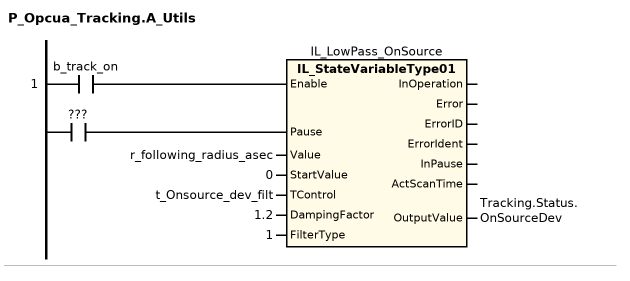
// NETWORK 1
IL_LowPass_OnSource(
    Enable := b_track_on,
    Value := r_following_radius_asec,
    StartValue := 0,
    TControl := t_Onsource_dev_filt,
    DampingFactor := 1.2,
    FilterType := 1,
    OutputValue => Tracking.Status.OnSourceDev); // IL_StateVariableType01
END_ACTION

END_PROGRAM

// IndraMotionMlc1/Application/POUs/OPCUA/OPCUA_Node/P_Opcua_Pointing
PROGRAM P_Opcua_Pointing
VAR
	TiltTemp_mV_1: LREAL;
	lr_one_x_off: LREAL;
	lr_one_y_off: LREAL;
	TiltTemp_mV_2: LREAL;
	lr_two_x_off: LREAL;
	lr_two_y_off: LREAL;
	IL_LowPass_Tilt_one_x: IL_StateVariableType01;
	IL_LowPass_Tilt_one_y: IL_StateVariableType01;
	IL_LowPass_Tilt_two_x: IL_StateVariableType01;
	IL_LowPass_Tilt_two_y: IL_StateVariableType01;
	t_one_x_filt_dt: TIME;
	t_one_y_filt_dt: TIME;
	t_two_x_filt_dt: TIME;
	t_two_y_filt_dt: TIME;
	b_tilt_filt_on: BOOL:= 1;
END_VAR

Pointing();
(*****Data*****)

(****************** Tilt Sensor **************************************)
// Tilt sensor one
Pointing.Status.TiltTemp_One := TiltTemp_mV_1*0.1;

lr_one_x_off:= (Pointing.TiltmeterParameters.One.x_zero+Pointing.TiltmeterParameters.One.x_zeroTC*Pointing.Status.TiltTemp_One)+
(Pointing.TiltmeterParameters.One.x_off+Pointing.TiltmeterParameters.One.x_offTC*Pointing.Status.TiltTemp_One);
lr_one_y_off:=(Pointing.TiltmeterParameters.One.y_zero+Pointing.TiltmeterParameters.One.y_zeroTC*Pointing.Status.TiltTemp_One)+
(Pointing.TiltmeterParameters.One.y_off+Pointing.TiltmeterParameters.One.y_offTC*Pointing.Status.TiltTemp_One);

Pointing.Status.TiltXArcsec_One:= Pointing.Status.TiltXRaw_mV_One*(Pointing.TiltmeterParameters.One.x_scale+Pointing.TiltmeterParameters.One.x_scaleTC*Pointing.Status.TiltTemp_One)+Pointing.TiltmeterParameters.One.x_off;
Pointing.Status.TiltYArcsec_One:= Pointing.Status.TiltYRaw_mV_One*(Pointing.TiltmeterParameters.One.y_scale+Pointing.TiltmeterParameters.One.y_scaleTC*Pointing.Status.TiltTemp_One)+Pointing.TiltmeterParameters.One.y_off;
t_one_x_filt_dt:= TO_TIME(Pointing.TiltmeterParameters.One.x_filt_dt*1000); //convert to milliseconds and TIME type.
t_one_y_filt_dt:= TO_TIME(Pointing.TiltmeterParameters.One.y_filt_dt*1000);

// Tilt Sensor Two
Pointing.Status.TiltTemp_Two := TiltTemp_mV_2*0.1;

lr_two_x_off:= (Pointing.TiltmeterParameters.Two.x_zero+Pointing.TiltmeterParameters.Two.x_zeroTC*Pointing.Status.TiltTemp_Two)+
(Pointing.TiltmeterParameters.Two.x_off+Pointing.TiltmeterParameters.Two.x_offTC*Pointing.Status.TiltTemp_Two);
lr_two_y_off:=(Pointing.TiltmeterParameters.Two.y_zero+Pointing.TiltmeterParameters.Two.y_zeroTC*Pointing.Status.TiltTemp_Two)+
(Pointing.TiltmeterParameters.Two.y_off+Pointing.TiltmeterParameters.Two.y_offTC*Pointing.Status.TiltTemp_Two);

Pointing.Status.TiltXArcsec_Two:= Pointing.Status.TiltXRaw_mV_Two*(Pointing.TiltmeterParameters.Two.x_scale+Pointing.TiltmeterParameters.Two.x_scaleTC*Pointing.Status.TiltTemp_Two)+Pointing.TiltmeterParameters.Two.x_off;
Pointing.Status.TiltYArcsec_Two:= Pointing.Status.TiltYRaw_mV_Two*(Pointing.TiltmeterParameters.Two.y_scale+Pointing.TiltmeterParameters.Two.y_scaleTC*Pointing.Status.TiltTemp_Two)+Pointing.TiltmeterParameters.Two.y_off;
t_two_x_filt_dt:= TO_TIME(Pointing.TiltmeterParameters.Two.x_filt_dt*1000); //convert to milliseconds and TIME type.
t_two_y_filt_dt:= TO_TIME(Pointing.TiltmeterParameters.Two.y_filt_dt*1000);

// Total point corrections

Pointing.Status.TotalPointCorr_Az:= Pointing.Status.StaticPmCorrVal_Az + Pointing.Status.TiltCorrVal_Az + Pointing.Status.AmbTempCorrVal_Az;
Pointing.Status.TotalPointCorr_El:= Pointing.Status.StaticPmCorrVal_El + Pointing.Status.TiltCorrVal_El + Pointing.Status.AmbTempCorrVal_El;

Pointing.Status.ActAmbTemp_East:= Pedestal_temp_EAST;  // These need to be checked
Pointing.Status.ActAmbTemp_South:= Pedestal_temp_SOUTH;;
Pointing.Status.ActAmbTemp_West:= Pedestal_temp_WEST;
//Pointing.Status.AmbTempCorrActive
//Pointing.Status.AmbTempCorrVal_Az
//Pointing.Status.AmbTempCorrVal_El
//Pointing.Status.BandForCorr
//Pointing.Status.StaticCorrActive
//Pointing.Status.StaticPmCorrVal_Az
//Pointing.Status.StaticPmCorrVal_El
//Pointing.Status.TiltCorrActive
//Pointing.Status.TiltCorrVal_Az
//Pointing.Status.TiltCorrVal_El
//Pointing.Status.TiltOne_On
//Pointing.Status.TiltTemp_One
//Pointing.Status.TiltTemp_Two
//Pointing.Status.TotalPointCorr_Az
//Pointing.Status.TotalPointCorr_El

ACTION A_Utils:
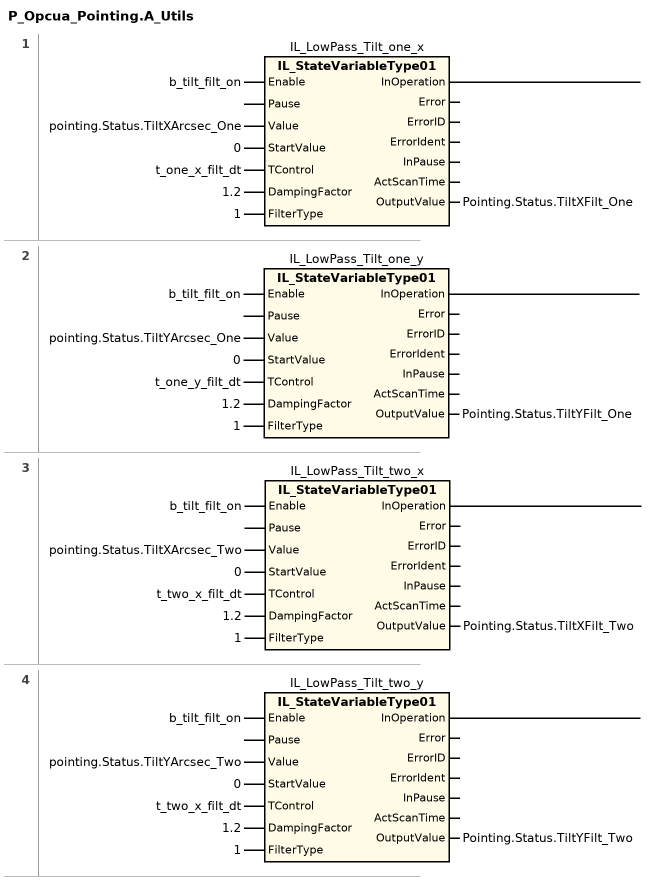
// NETWORK 1
IL_LowPass_Tilt_one_x(
    Enable := b_tilt_filt_on,
    Value := pointing.Status.TiltXArcsec_One,
    StartValue := 0,
    TControl := t_one_x_filt_dt,
    DampingFactor := 1.2,
    FilterType := 1,
    OutputValue => Pointing.Status.TiltXFilt_One); // IL_StateVariableType01

// NETWORK 2
IL_LowPass_Tilt_one_y(
    Enable := b_tilt_filt_on,
    Value := pointing.Status.TiltYArcsec_One,
    StartValue := 0,
    TControl := t_one_y_filt_dt,
    DampingFactor := 1.2,
    FilterType := 1,
    OutputValue => Pointing.Status.TiltYFilt_One); // IL_StateVariableType01

// NETWORK 3
IL_LowPass_Tilt_two_x(
    Enable := b_tilt_filt_on,
    Value := pointing.Status.TiltXArcsec_Two,
    StartValue := 0,
    TControl := t_two_x_filt_dt,
    DampingFactor := 1.2,
    FilterType := 1,
    OutputValue => Pointing.Status.TiltXFilt_Two); // IL_StateVariableType01

// NETWORK 4
IL_LowPass_Tilt_two_y(
    Enable := b_tilt_filt_on,
    Value := pointing.Status.TiltYArcsec_Two,
    StartValue := 0,
    TControl := t_two_x_filt_dt,
    DampingFactor := 1.2,
    FilterType := 1,
    OutputValue => Pointing.Status.TiltYFilt_Two); // IL_StateVariableType01
END_ACTION

END_PROGRAM

// IndraMotionMlc1/Application/POUs/Motion/Test_move
PROGRAM Test_move
VAR
	b_power: BOOL;
	b_enable_az1: BOOL;
	fb_enable_az1: MC_Power;
	b_enable_az1_done: BOOL;
	b_vel_az1: BOOL;
	fb_vel_az1: MC_MoveVelocity;
	vel_az1: REAL;
	b_enable_az2: BOOL;
	fb_enable_az2: MC_Power;
	b_enable_az2_done: BOOL;
	b_vel_az2: BOOL;
	vel_az2: REAL;
	fb_vel_az2: MC_MoveVelocity;
	b_enable_el1: BOOL;
	fb_enable_el1: MC_Power;
	b_enable_el1_done: BOOL;
	b_vel_el1: BOOL;
	vel_el1: REAL;
	fb_vel_el1: MC_MoveVelocity;
	b_vel_el2: BOOL;
	fb_vel_el2: MC_MoveVelocity;
	vel_el2: REAL;
	b_enable_el2: BOOL;
	fb_enable_el2: MC_Power;
	b_enable_FI1: BOOL;
	fb_enable_FI1: MC_Power;
	b_enable_el2_done: BOOL;
	b_enable_FI1_done: BOOL;
	b_vel_FI1: BOOL;
	fb_vel_FI1: MC_MoveVelocity;
	vel_FI1: REAL;
	b_enable_FI2: BOOL;
	fb_enable_FI2: MC_Power;
	b_enable_FI2_done: BOOL;
	b_vel_FI2: BOOL;
	vel_FI2: REAL;
	fb_vel_FI2: MC_MoveVelocity;
	b_torque_4: BOOL;
	b_torque_el2: BOOL;
	fb_torque_el2: MC_TorqueControl;
	b_torque_el2_done: BOOL;
	b_torque_az2: BOOL;
	fb_torque_az2: MC_TorqueControl;
	b_torque_az2_done: BOOL;
	fb_pos_az1: MC_MoveAbsolute;
	b_pos_az1: BOOL;
	pos_az1: REAL;
	b_stop_az: BOOL;
	fb_stop_AZ: MC_Stop;
	b_stop_el: BOOL;
	fb_stop_el: MC_Stop;
	b_pos_el1: BOOL;
	pos_el1: REAL;
	fb_pos_el1: MC_MoveAbsolute;
	b_pos_FI1: BOOL;
	pos_FI1: REAL;
	fb_pos_FI1: MC_MoveAbsolute;
	b_vel_1: BOOL;
	vel_1: REAL;
	fb_vel_1: MC_MoveVelocity;
	test_home_1: BOOL;
	fb_test_home: MB_Home;
	b_homeswitch_1: BOOL;
	b_torque_FI2: BOOL;
	fb_torque_FI2: MC_TorqueControl;
	b_torque_FI2_done: BOOL;
	b_touque_1: BOOL;
	fb_torque_az1: MC_TorqueControl;
	b_torque_az1_done: BOOL;
	torque_1: REAL;
	b_touque_3: BOOL;
	torque_3: REAL;
	fb_torque_el3: MC_TorqueControl;
END_VAR

(*IF r_pos_az>270.5 OR  r_pos_az<-270.5 THEN
			b_SCC_enable_on:=FALSE;
			b_SCC_enable_off:=TRUE; 
END_IF
*)




//axisdata[7].rActualPosition_i;
//test_move.power_move(); Commented out to prevent process using up resources.

ACTION power_move:
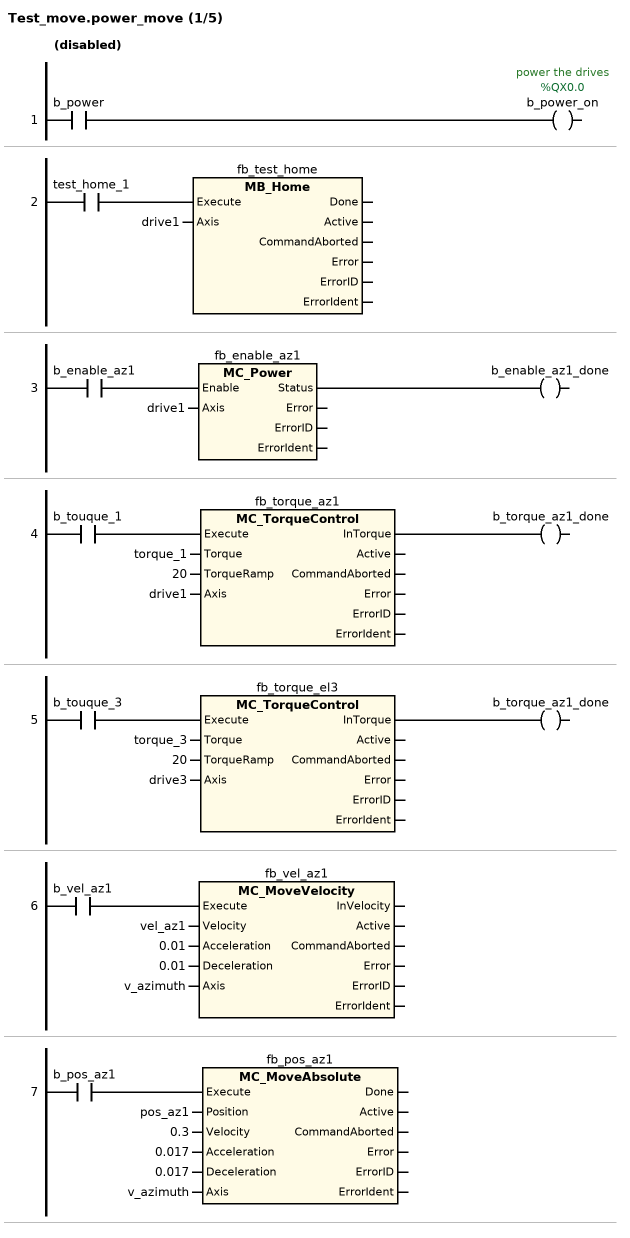
// NETWORK 1 (disabled)
//   b_power_on: power the drives | AT %QX0.0
// b_power_on := b_power;

// NETWORK 2
//   drive1: Real axis "Drive1" with axis number 1
fb_test_home(Execute := test_home_1, Axis := drive1); // MB_Home

// NETWORK 3
//   drive1: Real axis "Drive1" with axis number 1
fb_enable_az1(Enable := b_enable_az1, Axis := drive1); // MC_Power
b_enable_az1_done := fb_enable_az1.Status;

// NETWORK 4
//   drive1: Real axis "Drive4" with axis number 4
fb_torque_az1(Execute := b_touque_1, Torque := torque_1, TorqueRamp := 20, Axis := drive1); // MC_TorqueControl
b_torque_az1_done := fb_torque_az1.InTorque;

// NETWORK 5
//   drive3: Real axis "Drive4" with axis number 4
fb_torque_el3(Execute := b_touque_3, Torque := torque_3, TorqueRamp := 20, Axis := drive3); // MC_TorqueControl
b_torque_az1_done := fb_torque_el3.InTorque;

// NETWORK 6
//   v_azimuth: Virtual axis "v_azimuth" with axis number 7
fb_vel_az1(
    Execute := b_vel_az1,
    Velocity := vel_az1,
    Acceleration := 0.01,
    Deceleration := 0.01,
    Axis := v_azimuth); // MC_MoveVelocity

// NETWORK 7
//   v_azimuth: Virtual axis "v_azimuth" with axis number 7
fb_pos_az1(
    Execute := b_pos_az1,
    Position := pos_az1,
    Velocity := 0.3,
    Acceleration := 0.017,
    Deceleration := 0.017,
    Axis := v_azimuth); // MC_MoveAbsolute

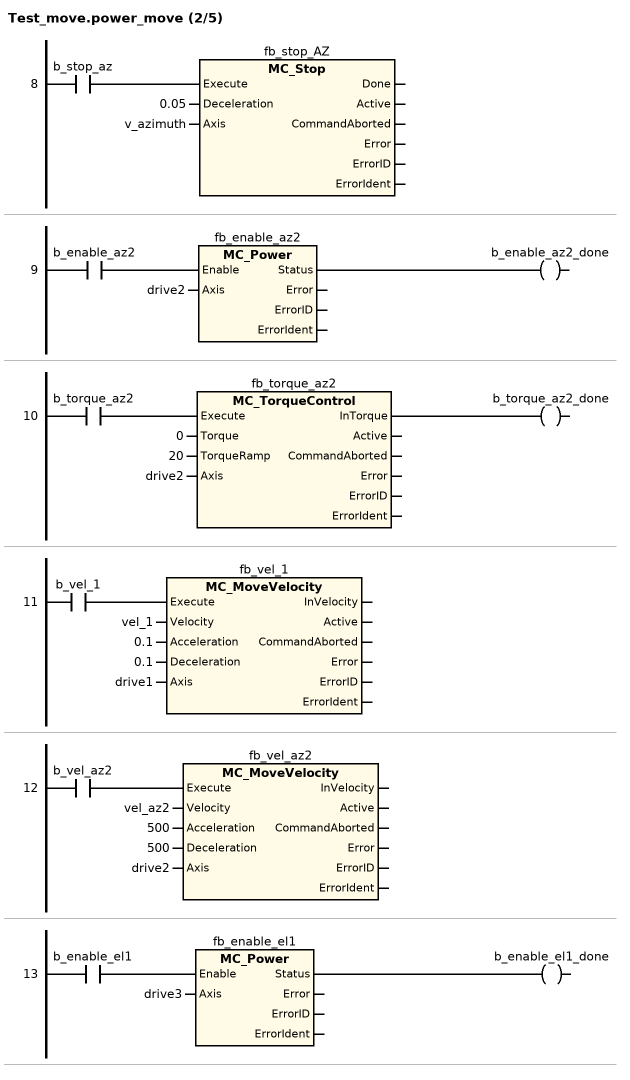
// NETWORK 8
//   v_azimuth: Virtual axis "v_azimuth" with axis number 7
fb_stop_AZ(Execute := b_stop_az, Deceleration := 0.05, Axis := v_azimuth); // MC_Stop

// NETWORK 9
//   drive2: Real axis "Drive2" with axis number 2
fb_enable_az2(Enable := b_enable_az2, Axis := drive2); // MC_Power
b_enable_az2_done := fb_enable_az2.Status;

// NETWORK 10
//   drive2: Real axis "Drive2" with axis number 2
fb_torque_az2(Execute := b_torque_az2, Torque := 0, TorqueRamp := 20, Axis := drive2); // MC_TorqueControl
b_torque_az2_done := fb_torque_az2.InTorque;

// NETWORK 11
//   drive1: Real axis "Drive1" with axis number 1
fb_vel_1(Execute := b_vel_1, Velocity := vel_1, Acceleration := 0.1, Deceleration := 0.1, Axis := drive1); // MC_MoveVelocity

// NETWORK 12
//   drive2: Real axis "Drive2" with axis number 2
fb_vel_az2(
    Execute := b_vel_az2,
    Velocity := vel_az2,
    Acceleration := 500,
    Deceleration := 500,
    Axis := drive2); // MC_MoveVelocity

// NETWORK 13
//   drive3: Real axis "Drive3" with axis number 3
fb_enable_el1(Enable := b_enable_el1, Axis := drive3); // MC_Power
b_enable_el1_done := fb_enable_el1.Status;

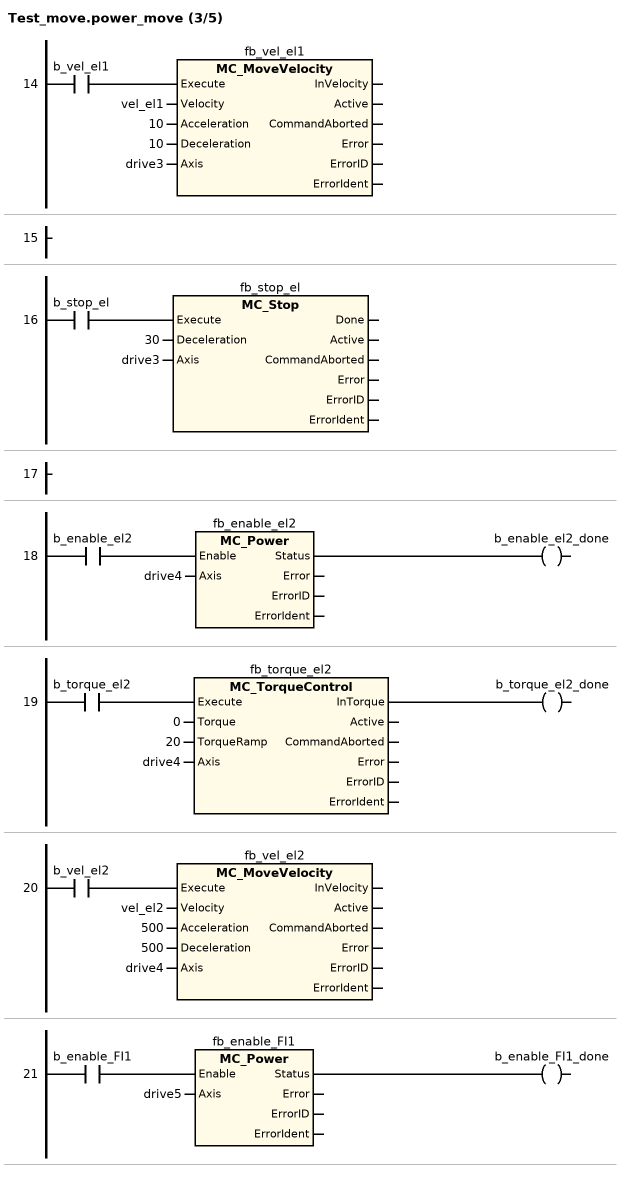
// NETWORK 14
//   drive3: Virtual axis "v_elevation" with axis number 8
fb_vel_el1(Execute := b_vel_el1, Velocity := vel_el1, Acceleration := 10, Deceleration := 10, Axis := drive3); // MC_MoveVelocity

// NETWORK 15

// NETWORK 16
//   drive3: Virtual axis "v_elevation" with axis number 8
fb_stop_el(Execute := b_stop_el, Deceleration := 30, Axis := drive3); // MC_Stop

// NETWORK 17

// NETWORK 18
//   drive4: Real axis "Drive4" with axis number 4
fb_enable_el2(Enable := b_enable_el2, Axis := drive4); // MC_Power
b_enable_el2_done := fb_enable_el2.Status;

// NETWORK 19
//   drive4: Real axis "Drive4" with axis number 4
fb_torque_el2(Execute := b_torque_el2, Torque := 0, TorqueRamp := 20, Axis := drive4); // MC_TorqueControl
b_torque_el2_done := fb_torque_el2.InTorque;

// NETWORK 20
//   drive4: Real axis "Drive4" with axis number 4
fb_vel_el2(
    Execute := b_vel_el2,
    Velocity := vel_el2,
    Acceleration := 500,
    Deceleration := 500,
    Axis := drive4); // MC_MoveVelocity

// NETWORK 21
//   drive5: Real axis "Drive5" with axis number 5
fb_enable_FI1(Enable := b_enable_FI1, Axis := drive5); // MC_Power
b_enable_FI1_done := fb_enable_FI1.Status;

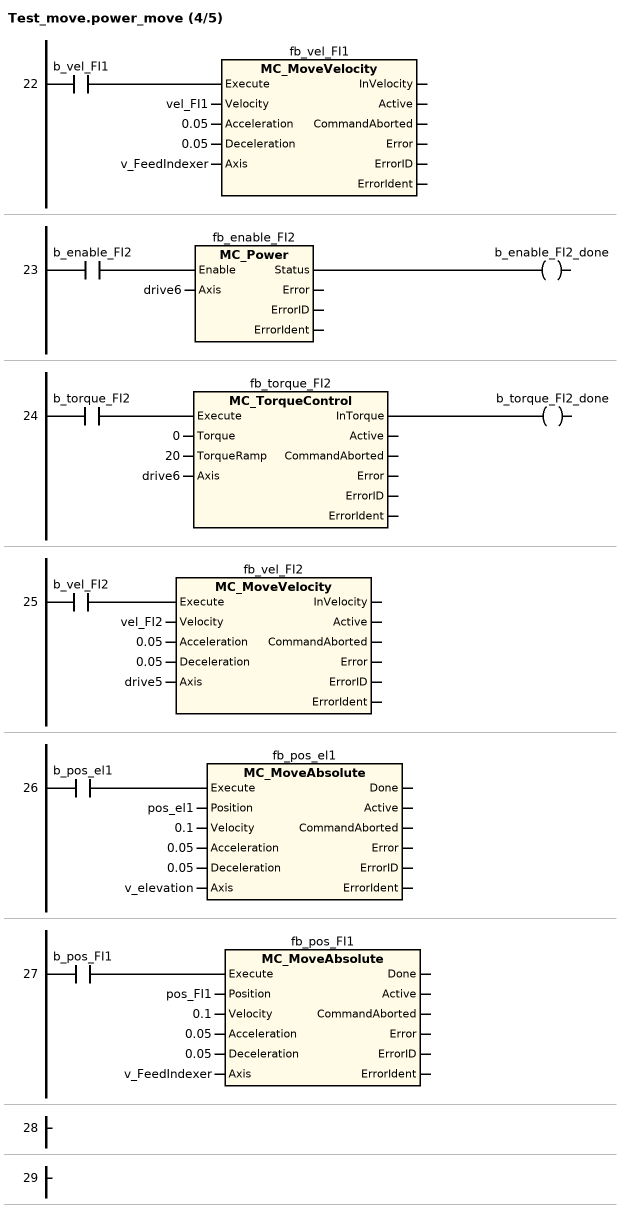
// NETWORK 22
//   v_FeedIndexer: Virtual axis "v_polarization" with axis number 9
fb_vel_FI1(
    Execute := b_vel_FI1,
    Velocity := vel_FI1,
    Acceleration := 0.05,
    Deceleration := 0.05,
    Axis := v_FeedIndexer); // MC_MoveVelocity

// NETWORK 23
//   drive6: Real axis "Drive6" with axis number 6
fb_enable_FI2(Enable := b_enable_FI2, Axis := drive6); // MC_Power
b_enable_FI2_done := fb_enable_FI2.Status;

// NETWORK 24
//   drive6: Real axis "Drive6" with axis number 6
fb_torque_FI2(Execute := b_torque_FI2, Torque := 0, TorqueRamp := 20, Axis := drive6); // MC_TorqueControl
b_torque_FI2_done := fb_torque_FI2.InTorque;

// NETWORK 25
//   drive5: Real axis "Drive5" with axis number 5
fb_vel_FI2(
    Execute := b_vel_FI2,
    Velocity := vel_FI2,
    Acceleration := 0.05,
    Deceleration := 0.05,
    Axis := drive5); // MC_MoveVelocity

// NETWORK 26
//   v_elevation: Virtual axis "v_elevation" with axis number 8
fb_pos_el1(
    Execute := b_pos_el1,
    Position := pos_el1,
    Velocity := 0.1,
    Acceleration := 0.05,
    Deceleration := 0.05,
    Axis := v_elevation); // MC_MoveAbsolute

// NETWORK 27
//   v_FeedIndexer: Virtual axis "v_polarization" with axis number 9
fb_pos_FI1(
    Execute := b_pos_FI1,
    Position := pos_FI1,
    Velocity := 0.1,
    Acceleration := 0.05,
    Deceleration := 0.05,
    Axis := v_FeedIndexer); // MC_MoveAbsolute

// NETWORK 28

// NETWORK 29

